   DATA[560,19] := 2.0;
   DATA[560,20] := 148.808;
   DATA[560,21] := 156.0369;
   DATA[560,22] := 1.722487;
   DATA[560,23] := 988.6696;
   DATA[560,24] := 2.0;
   DATA[560,25] := 2.0;
   DATA[560,26] := 7.880544;
   DATA[560,27] := 144.7578;
   DATA[560,28] := 263.4581;
   DATA[560,29] := 12.07383;
   DATA[560,30] := 1.731479;
   DATA[560,31] := 1.287306;
   DATA[560,32] := 0.7353967;
   DATA[560,33] := 0.3080421;
   DATA[560,34] := 2.0;
   DATA[560,35] := 251.2977;
   DATA[560,36] := 1.746067;
   DATA[560,37] := 190.0474;
   DATA[560,38] := 0.000128152;
   DATA[560,39] := 1.0;
   DATA[561,0] := 2.621785;
   DATA[561,1] := 530.344;
   DATA[561,2] := 2.0;
   DATA[561,3] := 2.0;
   DATA[561,4] := 262.1764;
   DATA[561,5] := 8.395475;
   DATA[561,6] := 327.9159;
   DATA[561,7] := 2.4427;
   DATA[561,8] := 2.0;
   DATA[561,9] := 2.0;
   DATA[561,10] := 2.0;
   DATA[561,11] := 19.66835;
   DATA[561,12] := 2.211959;
   DATA[561,13] := 981.4791;
   DATA[561,14] := 1.0;
   DATA[561,15] := 2.0;
   DATA[561,16] := 1.0;
   DATA[561,17] := 1.0;
   DATA[561,18] := 1.0;
   DATA[561,19] := 2.0;
   DATA[561,20] := 148.808;
   DATA[561,21] := 156.0369;
   DATA[561,22] := 1.72159;
   DATA[561,23] := 988.7465;
   DATA[561,24] := 2.0;
   DATA[561,25] := 2.0;
   DATA[561,26] := 7.880544;
   DATA[561,27] := 144.7578;
   DATA[561,28] := 263.4261;
   DATA[561,29] := 12.07383;
   DATA[561,30] := 1.731479;
   DATA[561,31] := 1.274625;
   DATA[561,32] := 0.7353967;
   DATA[561,33] := 0.3087468;
   DATA[561,34] := 2.0;
   DATA[561,35] := 251.2977;
   DATA[561,36] := 1.746067;
   DATA[561,37] := 190.0474;
   DATA[561,38] := 0.000128152;
   DATA[561,39] := 1.0;
   DATA[562,0] := 2.61634;
   DATA[562,1] := 531.9534;
   DATA[562,2] := 2.0;
   DATA[562,3] := 2.0;
   DATA[562,4] := 262.1764;
   DATA[562,5] := 8.395475;
   DATA[562,6] := 327.9159;
   DATA[562,7] := 2.4427;
   DATA[562,8] := 2.0;
   DATA[562,9] := 2.0;
   DATA[562,10] := 2.0;
   DATA[562,11] := 19.66835;
   DATA[562,12] := 2.214906;
   DATA[562,13] := 981.4391;
   DATA[562,14] := 1.0;
   DATA[562,15] := 2.0;
   DATA[562,16] := 1.0;
   DATA[562,17] := 1.0;
   DATA[562,18] := 1.0;
   DATA[562,19] := 2.0;
   DATA[562,20] := 148.808;
   DATA[562,21] := 156.0369;
   DATA[562,22] := 1.718515;
   DATA[562,23] := 989.0925;
   DATA[562,24] := 2.0;
   DATA[562,25] := 2.0;
   DATA[562,26] := 7.880544;
   DATA[562,27] := 144.7578;
   DATA[562,28] := 263.4261;
   DATA[562,29] := 12.07383;
   DATA[562,30] := 1.731479;
   DATA[562,31] := 1.261432;
   DATA[562,32] := 0.7353967;
   DATA[562,33] := 0.3068891;
   DATA[562,34] := 2.0;
   DATA[562,35] := 251.0734;
   DATA[562,36] := 1.746067;
   DATA[562,37] := 189.727;
   DATA[562,38] := 0.000128152;
   DATA[562,39] := 1.0;
   DATA[563,0] := 2.6157;
   DATA[563,1] := 532.5422;
   DATA[563,2] := 2.0;
   DATA[563,3] := 2.0;
   DATA[563,4] := 262.1764;
   DATA[563,5] := 8.395155;
   DATA[563,6] := 327.9159;
   DATA[563,7] := 2.4427;
   DATA[563,8] := 2.0;
   DATA[563,9] := 2.0;
   DATA[563,10] := 2.0;
   DATA[563,11] := 19.66835;
   DATA[563,12] := 2.214906;
   DATA[563,13] := 981.5593;
   DATA[563,14] := 1.0;
   DATA[563,15] := 2.0;
   DATA[563,16] := 1.0;
   DATA[563,17] := 1.0;
   DATA[563,18] := 1.0;
   DATA[563,19] := 2.0;
   DATA[563,20] := 148.808;
   DATA[563,21] := 156.0369;
   DATA[563,22] := 1.718515;
   DATA[563,23] := 988.708;
   DATA[563,24] := 2.0;
   DATA[563,25] := 2.0;
   DATA[563,26] := 7.880544;
   DATA[563,27] := 144.7578;
   DATA[563,28] := 263.4261;
   DATA[563,29] := 12.07383;
   DATA[563,30] := 1.731479;
   DATA[563,31] := 1.25554;
   DATA[563,32] := 0.7353967;
   DATA[563,33] := 0.3066329;
   DATA[563,34] := 2.0;
   DATA[563,35] := 251.0734;
   DATA[563,36] := 1.746067;
   DATA[563,37] := 189.727;
   DATA[563,38] := 0.000128152;
   DATA[563,39] := 1.0;
   DATA[564,0] := 2.593601;
   DATA[564,1] := 532.8954;
   DATA[564,2] := 2.0;
   DATA[564,3] := 2.0;
   DATA[564,4] := 262.1764;
   DATA[564,5] := 8.394835;
   DATA[564,6] := 327.9159;
   DATA[564,7] := 2.444879;
   DATA[564,8] := 2.0;
   DATA[564,9] := 2.0;
   DATA[564,10] := 2.0;
   DATA[564,11] := 19.66835;
   DATA[564,12] := 2.21324;
   DATA[564,13] := 980.8383;
   DATA[564,14] := 1.0;
   DATA[564,15] := 2.0;
   DATA[564,16] := 1.0;
   DATA[564,17] := 1.0;
   DATA[564,18] := 1.0;
   DATA[564,19] := 2.0;
   DATA[564,20] := 148.808;
   DATA[564,21] := 156.0369;
   DATA[564,22] := 1.718515;
   DATA[564,23] := 989.0925;
   DATA[564,24] := 2.0;
   DATA[564,25] := 2.0;
   DATA[564,26] := 7.880544;
   DATA[564,27] := 144.7578;
   DATA[564,28] := 263.4261;
   DATA[564,29] := 12.07383;
   DATA[564,30] := 1.7293;
   DATA[564,31] := 1.254643;
   DATA[564,32] := 0.7353967;
   DATA[564,33] := 0.3065048;
   DATA[564,34] := 2.0;
   DATA[564,35] := 250.9773;
   DATA[564,36] := 1.746067;
   DATA[564,37] := 189.727;
   DATA[564,38] := 0.000128152;
   DATA[564,39] := 1.0;
   DATA[565,0] := 2.572142;
   DATA[565,1] := 532.9739;
   DATA[565,2] := 2.0;
   DATA[565,3] := 2.0;
   DATA[565,4] := 262.1764;
   DATA[565,5] := 8.394835;
   DATA[565,6] := 327.9159;
   DATA[565,7] := 2.444879;
   DATA[565,8] := 2.0;
   DATA[565,9] := 2.0;
   DATA[565,10] := 2.0;
   DATA[565,11] := 19.67796;
   DATA[565,12] := 2.21324;
   DATA[565,13] := 981.1587;
   DATA[565,14] := 1.0;
   DATA[565,15] := 2.0;
   DATA[565,16] := 1.0;
   DATA[565,17] := 1.0;
   DATA[565,18] := 1.0;
   DATA[565,19] := 2.0;
   DATA[565,20] := 148.808;
   DATA[565,21] := 156.0369;
   DATA[565,22] := 1.718515;
   DATA[565,23] := 988.9387;
   DATA[565,24] := 2.0;
   DATA[565,25] := 2.0;
   DATA[565,26] := 7.880544;
   DATA[565,27] := 144.7578;
   DATA[565,28] := 263.4261;
   DATA[565,29] := 12.07383;
   DATA[565,30] := 1.7293;
   DATA[565,31] := 1.268989;
   DATA[565,32] := 0.7353967;
   DATA[565,33] := 0.3065048;
   DATA[565,34] := 2.0;
   DATA[565,35] := 250.9132;
   DATA[565,36] := 1.746067;
   DATA[565,37] := 189.5988;
   DATA[565,38] := 0.000128152;
   DATA[565,39] := 1.0;
   DATA[566,0] := 2.560933;
   DATA[566,1] := 532.8562;
   DATA[566,2] := 2.0;
   DATA[566,3] := 2.0;
   DATA[566,4] := 262.1764;
   DATA[566,5] := 8.394835;
   DATA[566,6] := 327.9159;
   DATA[566,7] := 2.444879;
   DATA[566,8] := 2.0;
   DATA[566,9] := 2.0;
   DATA[566,10] := 2.0;
   DATA[566,11] := 19.67796;
   DATA[566,12] := 2.21324;
   DATA[566,13] := 981.1987;
   DATA[566,14] := 1.0;
   DATA[566,15] := 2.0;
   DATA[566,16] := 1.0;
   DATA[566,17] := 1.0;
   DATA[566,18] := 1.0;
   DATA[566,19] := 2.0;
   DATA[566,20] := 148.808;
   DATA[566,21] := 156.0369;
   DATA[566,22] := 1.717105;
   DATA[566,23] := 988.4773;
   DATA[566,24] := 2.0;
   DATA[566,25] := 2.0;
   DATA[566,26] := 7.880544;
   DATA[566,27] := 144.7578;
   DATA[566,28] := 263.4261;
   DATA[566,29] := 12.07383;
   DATA[566,30] := 1.726096;
   DATA[566,31] := 1.271039;
   DATA[566,32] := 0.736421;
   DATA[566,33] := 0.3065048;
   DATA[566,34] := 2.0;
   DATA[566,35] := 250.5928;
   DATA[566,36] := 1.665972;
   DATA[566,37] := 189.5347;
   DATA[566,38] := 0.000128152;
   DATA[566,39] := 1.0;
   DATA[567,0] := 2.542036;
   DATA[567,1] := 532.7384;
   DATA[567,2] := 2.0;
   DATA[567,3] := 2.0;
   DATA[567,4] := 262.1764;
   DATA[567,5] := 8.394835;
   DATA[567,6] := 327.9159;
   DATA[567,7] := 2.442444;
   DATA[567,8] := 2.0;
   DATA[567,9] := 2.0;
   DATA[567,10] := 2.0;
   DATA[567,11] := 19.67796;
   DATA[567,12] := 2.21324;
   DATA[567,13] := 981.1587;
   DATA[567,14] := 1.0;
   DATA[567,15] := 2.0;
   DATA[567,16] := 1.0;
   DATA[567,17] := 1.0;
   DATA[567,18] := 1.0;
   DATA[567,19] := 2.0;
   DATA[567,20] := 148.808;
   DATA[567,21] := 156.0369;
   DATA[567,22] := 1.716592;
   DATA[567,23] := 989.0541;
   DATA[567,24] := 2.0;
   DATA[567,25] := 2.0;
   DATA[567,26] := 7.880544;
   DATA[567,27] := 144.8859;
   DATA[567,28] := 263.4261;
   DATA[567,29] := 12.07383;
   DATA[567,30] := 1.726096;
   DATA[567,31] := 1.280261;
   DATA[567,32] := 0.7370611;
   DATA[567,33] := 0.3065048;
   DATA[567,34] := 2.0;
   DATA[567,35] := 250.5928;
   DATA[567,36] := 1.665972;
   DATA[567,37] := 189.5027;
   DATA[567,38] := 0.000128152;
   DATA[567,39] := 1.0;
   DATA[568,0] := 2.530506;
   DATA[568,1] := 532.4637;
   DATA[568,2] := 2.0;
   DATA[568,3] := 2.0;
   DATA[568,4] := 262.1764;
   DATA[568,5] := 8.394835;
   DATA[568,6] := 327.9159;
   DATA[568,7] := 2.441162;
   DATA[568,8] := 2.0;
   DATA[568,9] := 2.0;
   DATA[568,10] := 2.0;
   DATA[568,11] := 19.63954;
   DATA[568,12] := 2.211318;
   DATA[568,13] := 980.9985;
   DATA[568,14] := 1.0;
   DATA[568,15] := 2.0;
   DATA[568,16] := 1.0;
   DATA[568,17] := 1.0;
   DATA[568,18] := 1.0;
   DATA[568,19] := 2.0;
   DATA[568,20] := 148.808;
   DATA[568,21] := 156.0369;
   DATA[568,22] := 1.716592;
   DATA[568,23] := 988.708;
   DATA[568,24] := 2.0;
   DATA[568,25] := 2.0;
   DATA[568,26] := 7.880544;
   DATA[568,27] := 144.9116;
   DATA[568,28] := 263.4261;
   DATA[568,29] := 12.07383;
   DATA[568,30] := 1.726096;
   DATA[568,31] := 1.290124;
   DATA[568,32] := 0.7370611;
   DATA[568,33] := 0.3083624;
   DATA[568,34] := 2.0;
   DATA[568,35] := 250.5928;
   DATA[568,36] := 1.665972;
   DATA[568,37] := 189.5027;
   DATA[568,38] := 0.000128152;
   DATA[568,39] := 1.0;
   DATA[569,0] := 2.510649;
   DATA[569,1] := 532.2674;
   DATA[569,2] := 2.0;
   DATA[569,3] := 2.0;
   DATA[569,4] := 262.1764;
   DATA[569,5] := 8.394835;
   DATA[569,6] := 327.9159;
   DATA[569,7] := 2.440521;
   DATA[569,8] := 2.0;
   DATA[569,9] := 2.0;
   DATA[569,10] := 2.0;
   DATA[569,11] := 19.63954;
   DATA[569,12] := 2.210294;
   DATA[569,13] := 980.638;
   DATA[569,14] := 1.0;
   DATA[569,15] := 2.0;
   DATA[569,16] := 1.0;
   DATA[569,17] := 1.0;
   DATA[569,18] := 1.0;
   DATA[569,19] := 2.0;
   DATA[569,20] := 148.808;
   DATA[569,21] := 156.0369;
   DATA[569,22] := 1.717746;
   DATA[569,23] := 988.8618;
   DATA[569,24] := 2.0;
   DATA[569,25] := 2.0;
   DATA[569,26] := 7.880544;
   DATA[569,27] := 144.9116;
   DATA[569,28] := 263.4261;
   DATA[569,29] := 12.07383;
   DATA[569,30] := 1.726096;
   DATA[569,31] := 1.291277;
   DATA[569,32] := 0.7370611;
   DATA[569,33] := 0.3083624;
   DATA[569,34] := 2.0;
   DATA[569,35] := 250.8171;
   DATA[569,36] := 1.665972;
   DATA[569,37] := 189.5027;
   DATA[569,38] := 0.000128152;
   DATA[569,39] := 1.0;
   DATA[570,0] := 2.498799;
   DATA[570,1] := 532.3459;
   DATA[570,2] := 2.0;
   DATA[570,3] := 2.0;
   DATA[570,4] := 262.1764;
   DATA[570,5] := 8.394835;
   DATA[570,6] := 327.9159;
   DATA[570,7] := 2.439881;
   DATA[570,8] := 2.0;
   DATA[570,9] := 2.0;
   DATA[570,10] := 2.0;
   DATA[570,11] := 19.63954;
   DATA[570,12] := 2.210294;
   DATA[570,13] := 980.598;
   DATA[570,14] := 1.0;
   DATA[570,15] := 2.0;
   DATA[570,16] := 1.0;
   DATA[570,17] := 1.0;
   DATA[570,18] := 1.0;
   DATA[570,19] := 2.0;
   DATA[570,20] := 148.808;
   DATA[570,21] := 156.0369;
   DATA[570,22] := 1.717746;
   DATA[570,23] := 988.8618;
   DATA[570,24] := 2.0;
   DATA[570,25] := 2.0;
   DATA[570,26] := 7.880544;
   DATA[570,27] := 144.9116;
   DATA[570,28] := 263.4261;
   DATA[570,29] := 12.07383;
   DATA[570,30] := 1.726096;
   DATA[570,31] := 1.286025;
   DATA[570,32] := 0.7359089;
   DATA[570,33] := 0.3083624;
   DATA[570,34] := 2.0;
   DATA[570,35] := 250.8652;
   DATA[570,36] := 1.665972;
   DATA[570,37] := 189.5027;
   DATA[570,38] := 0.000128152;
   DATA[570,39] := 1.0;
   DATA[571,0] := 2.484066;
   DATA[571,1] := 532.1497;
   DATA[571,2] := 2.0;
   DATA[571,3] := 2.0;
   DATA[571,4] := 262.1764;
   DATA[571,5] := 8.394835;
   DATA[571,6] := 327.9159;
   DATA[571,7] := 2.439881;
   DATA[571,8] := 2.0;
   DATA[571,9] := 2.0;
   DATA[571,10] := 2.0;
   DATA[571,11] := 19.65875;
   DATA[571,12] := 2.214777;
   DATA[571,13] := 980.638;
   DATA[571,14] := 1.0;
   DATA[571,15] := 2.0;
   DATA[571,16] := 1.0;
   DATA[571,17] := 1.0;
   DATA[571,18] := 1.0;
   DATA[571,19] := 2.0;
   DATA[571,20] := 148.808;
   DATA[571,21] := 156.0369;
   DATA[571,22] := 1.717746;
   DATA[571,23] := 989.4386;
   DATA[571,24] := 2.0;
   DATA[571,25] := 2.0;
   DATA[571,26] := 7.880544;
   DATA[571,27] := 144.9116;
   DATA[571,28] := 263.4261;
   DATA[571,29] := 12.07383;
   DATA[571,30] := 1.726096;
   DATA[571,31] := 1.287947;
   DATA[571,32] := 0.7347566;
   DATA[571,33] := 0.3083624;
   DATA[571,34] := 2.0;
   DATA[571,35] := 250.9453;
   DATA[571,36] := 1.665972;
   DATA[571,37] := 189.743;
   DATA[571,38] := 0.000128152;
   DATA[571,39] := 1.0;
   DATA[572,0] := 2.475098;
   DATA[572,1] := 532.0711;
   DATA[572,2] := 2.0;
   DATA[572,3] := 2.0;
   DATA[572,4] := 262.1764;
   DATA[572,5] := 8.394835;
   DATA[572,6] := 327.9159;
   DATA[572,7] := 2.439881;
   DATA[572,8] := 2.0;
   DATA[572,9] := 2.0;
   DATA[572,10] := 2.0;
   DATA[572,11] := 19.65875;
   DATA[572,12] := 2.214777;
   DATA[572,13] := 980.5579;
   DATA[572,14] := 1.0;
   DATA[572,15] := 2.0;
   DATA[572,16] := 1.0;
   DATA[572,17] := 1.0;
   DATA[572,18] := 1.0;
   DATA[572,19] := 2.0;
   DATA[572,20] := 148.808;
   DATA[572,21] := 155.8575;
   DATA[572,22] := 1.717746;
   DATA[572,23] := 989.131;
   DATA[572,24] := 2.0;
   DATA[572,25] := 2.0;
   DATA[572,26] := 7.880544;
   DATA[572,27] := 144.9116;
   DATA[572,28] := 263.4261;
   DATA[572,29] := 12.07383;
   DATA[572,30] := 1.726352;
   DATA[572,31] := 1.272064;
   DATA[572,32] := 0.7347566;
   DATA[572,33] := 0.3083624;
   DATA[572,34] := 2.0;
   DATA[572,35] := 250.9453;
   DATA[572,36] := 1.665972;
   DATA[572,37] := 189.743;
   DATA[572,38] := 0.000128152;
   DATA[572,39] := 1.0;
   DATA[573,0] := 2.462287;
   DATA[573,1] := 531.7964;
   DATA[573,2] := 2.0;
   DATA[573,3] := 2.0;
   DATA[573,4] := 262.1764;
   DATA[573,5] := 8.394835;
   DATA[573,6] := 327.9159;
   DATA[573,7] := 2.439881;
   DATA[573,8] := 2.0;
   DATA[573,9] := 2.0;
   DATA[573,10] := 2.0;
   DATA[573,11] := 19.70037;
   DATA[573,12] := 2.21324;
   DATA[573,13] := 980.7982;
   DATA[573,14] := 1.0;
   DATA[573,15] := 2.0;
   DATA[573,16] := 1.0;
   DATA[573,17] := 1.0;
   DATA[573,18] := 1.0;
   DATA[573,19] := 2.0;
   DATA[573,20] := 148.808;
   DATA[573,21] := 155.8575;
   DATA[573,22] := 1.717746;
   DATA[573,23] := 989.4001;
   DATA[573,24] := 2.0;
   DATA[573,25] := 2.0;
   DATA[573,26] := 7.880544;
   DATA[573,27] := 144.9116;
   DATA[573,28] := 263.4261;
   DATA[573,29] := 12.07383;
   DATA[573,30] := 1.726737;
   DATA[573,31] := 1.280005;
   DATA[573,32] := 0.7347566;
   DATA[573,33] := 0.3083624;
   DATA[573,34] := 2.0;
   DATA[573,35] := 250.9453;
   DATA[573,36] := 1.665972;
   DATA[573,37] := 189.743;
   DATA[573,38] := 0.000128152;
   DATA[573,39] := 1.0;
   DATA[574,0] := 2.449476;
   DATA[574,1] := 531.9141;
   DATA[574,2] := 2.0;
   DATA[574,3] := 2.0;
   DATA[574,4] := 262.1764;
   DATA[574,5] := 8.394835;
   DATA[574,6] := 327.839;
   DATA[574,7] := 2.442188;
   DATA[574,8] := 2.0;
   DATA[574,9] := 2.0;
   DATA[574,10] := 2.0;
   DATA[574,11] := 19.70037;
   DATA[574,12] := 2.212215;
   DATA[574,13] := 980.7982;
   DATA[574,14] := 1.0;
   DATA[574,15] := 2.0;
   DATA[574,16] := 1.0;
   DATA[574,17] := 1.0;
   DATA[574,18] := 1.0;
   DATA[574,19] := 2.0;
   DATA[574,20] := 148.808;
   DATA[574,21] := 155.8575;
   DATA[574,22] := 1.717746;
   DATA[574,23] := 989.3232;
   DATA[574,24] := 2.0;
   DATA[574,25] := 2.0;
   DATA[574,26] := 7.880544;
   DATA[574,27] := 144.9116;
   DATA[574,28] := 263.4261;
   DATA[574,29] := 12.07383;
   DATA[574,30] := 1.726737;
   DATA[574,31] := 1.291405;
   DATA[574,32] := 0.7347566;
   DATA[574,33] := 0.3083624;
   DATA[574,34] := 2.0;
   DATA[574,35] := 250.9453;
   DATA[574,36] := 1.665972;
   DATA[574,37] := 189.743;
   DATA[574,38] := 0.000128152;
   DATA[574,39] := 1.0;
   DATA[575,0] := 2.433142;
   DATA[575,1] := 532.1889;
   DATA[575,2] := 2.0;
   DATA[575,3] := 2.0;
   DATA[575,4] := 262.1764;
   DATA[575,5] := 8.394835;
   DATA[575,6] := 327.839;
   DATA[575,7] := 2.442188;
   DATA[575,8] := 2.0;
   DATA[575,9] := 2.0;
   DATA[575,10] := 2.0;
   DATA[575,11] := 19.73878;
   DATA[575,12] := 2.212215;
   DATA[575,13] := 980.678;
   DATA[575,14] := 1.0;
   DATA[575,15] := 2.0;
   DATA[575,16] := 1.0;
   DATA[575,17] := 1.0;
   DATA[575,18] := 1.0;
   DATA[575,19] := 2.0;
   DATA[575,20] := 148.808;
   DATA[575,21] := 155.678;
   DATA[575,22] := 1.717746;
   DATA[575,23] := 989.4771;
   DATA[575,24] := 2.0;
   DATA[575,25] := 2.0;
   DATA[575,26] := 7.880544;
   DATA[575,27] := 144.9116;
   DATA[575,28] := 263.4261;
   DATA[575,29] := 12.07383;
   DATA[575,30] := 1.728531;
   DATA[575,31] := 1.291405;
   DATA[575,32] := 0.7355248;
   DATA[575,33] := 0.3083624;
   DATA[575,34] := 2.0;
   DATA[575,35] := 250.9773;
   DATA[575,36] := 1.665972;
   DATA[575,37] := 189.743;
   DATA[575,38] := 0.000128152;
   DATA[575,39] := 1.0;
   DATA[576,0] := 2.428979;
   DATA[576,1] := 532.3459;
   DATA[576,2] := 2.0;
   DATA[576,3] := 2.0;
   DATA[576,4] := 262.1764;
   DATA[576,5] := 8.394835;
   DATA[576,6] := 327.839;
   DATA[576,7] := 2.442188;
   DATA[576,8] := 2.0;
   DATA[576,9] := 2.0;
   DATA[576,10] := 2.0;
   DATA[576,11] := 19.74838;
   DATA[576,12] := 2.21055;
   DATA[576,13] := 980.598;
   DATA[576,14] := 1.0;
   DATA[576,15] := 2.0;
   DATA[576,16] := 1.0;
   DATA[576,17] := 1.0;
   DATA[576,18] := 1.0;
   DATA[576,19] := 2.0;
   DATA[576,20] := 148.808;
   DATA[576,21] := 155.678;
   DATA[576,22] := 1.717746;
   DATA[576,23] := 989.5155;
   DATA[576,24] := 2.0;
   DATA[576,25] := 2.0;
   DATA[576,26] := 7.880544;
   DATA[576,27] := 144.9116;
   DATA[576,28] := 263.4261;
   DATA[576,29] := 12.07383;
   DATA[576,30] := 1.728531;
   DATA[576,31] := 1.291405;
   DATA[576,32] := 0.7355248;
   DATA[576,33] := 0.3083624;
   DATA[576,34] := 2.0;
   DATA[576,35] := 250.9933;
   DATA[576,36] := 1.665972;
   DATA[576,37] := 189.743;
   DATA[576,38] := 0.000128152;
   DATA[576,39] := 1.0;
   DATA[577,0] := 2.428979;
   DATA[577,1] := 532.6992;
   DATA[577,2] := 2.0;
   DATA[577,3] := 2.0;
   DATA[577,4] := 262.1764;
   DATA[577,5] := 8.394835;
   DATA[577,6] := 327.839;
   DATA[577,7] := 2.442188;
   DATA[577,8] := 2.0;
   DATA[577,9] := 2.0;
   DATA[577,10] := 2.0;
   DATA[577,11] := 19.74838;
   DATA[577,12] := 2.209525;
   DATA[577,13] := 980.7582;
   DATA[577,14] := 1.0;
   DATA[577,15] := 2.0;
   DATA[577,16] := 1.0;
   DATA[577,17] := 1.0;
   DATA[577,18] := 1.0;
   DATA[577,19] := 2.0;
   DATA[577,20] := 148.808;
   DATA[577,21] := 155.678;
   DATA[577,22] := 1.717746;
   DATA[577,23] := 989.7847;
   DATA[577,24] := 2.0;
   DATA[577,25] := 2.0;
   DATA[577,26] := 7.880544;
   DATA[577,27] := 144.9116;
   DATA[577,28] := 263.3299;
   DATA[577,29] := 12.07383;
   DATA[577,30] := 1.728531;
   DATA[577,31] := 1.280902;
   DATA[577,32] := 0.7355248;
   DATA[577,33] := 0.3083624;
   DATA[577,34] := 2.0;
   DATA[577,35] := 250.9933;
   DATA[577,36] := 1.665972;
   DATA[577,37] := 189.743;
   DATA[577,38] := 0.000128152;
   DATA[577,39] := 1.0;
   DATA[578,0] := 2.458444;
   DATA[578,1] := 532.7384;
   DATA[578,2] := 2.0;
   DATA[578,3] := 2.0;
   DATA[578,4] := 262.1764;
   DATA[578,5] := 8.394835;
   DATA[578,6] := 327.839;
   DATA[578,7] := 2.44411;
   DATA[578,8] := 2.0;
   DATA[578,9] := 2.0;
   DATA[578,10] := 2.0;
   DATA[578,11] := 19.74838;
   DATA[578,12] := 2.207475;
   DATA[578,13] := 980.8383;
   DATA[578,14] := 1.0;
   DATA[578,15] := 2.0;
   DATA[578,16] := 1.0;
   DATA[578,17] := 1.0;
   DATA[578,18] := 1.0;
   DATA[578,19] := 2.0;
   DATA[578,20] := 148.808;
   DATA[578,21] := 155.678;
   DATA[578,22] := 1.717746;
   DATA[578,23] := 989.8616;
   DATA[578,24] := 2.0;
   DATA[578,25] := 2.0;
   DATA[578,26] := 7.880544;
   DATA[578,27] := 144.9116;
   DATA[578,28] := 263.3299;
   DATA[578,29] := 12.07383;
   DATA[578,30] := 1.728531;
   DATA[578,31] := 1.263097;
   DATA[578,32] := 0.7355248;
   DATA[578,33] := 0.3083624;
   DATA[578,34] := 2.0;
   DATA[578,35] := 250.9933;
   DATA[578,36] := 1.665972;
   DATA[578,37] := 189.743;
   DATA[578,38] := 0.000128152;
   DATA[578,39] := 1.0;
   DATA[579,0] := 2.495596;
   DATA[579,1] := 533.3272;
   DATA[579,2] := 2.0;
   DATA[579,3] := 2.0;
   DATA[579,4] := 262.1764;
   DATA[579,5] := 8.394835;
   DATA[579,6] := 327.839;
   DATA[579,7] := 2.442956;
   DATA[579,8] := 2.0;
   DATA[579,9] := 2.0;
   DATA[579,10] := 2.0;
   DATA[579,11] := 19.74838;
   DATA[579,12] := 2.206066;
   DATA[579,13] := 981.0786;
   DATA[579,14] := 1.0;
   DATA[579,15] := 2.0;
   DATA[579,16] := 1.0;
   DATA[579,17] := 1.0;
   DATA[579,18] := 1.0;
   DATA[579,19] := 2.0;
   DATA[579,20] := 148.808;
   DATA[579,21] := 155.678;
   DATA[579,22] := 1.715952;
   DATA[579,23] := 989.7847;
   DATA[579,24] := 2.0;
   DATA[579,25] := 2.0;
   DATA[579,26] := 7.880544;
   DATA[579,27] := 144.9116;
   DATA[579,28] := 263.3299;
   DATA[579,29] := 12.07383;
   DATA[579,30] := 1.728531;
   DATA[579,31] := 1.261816;
   DATA[579,32] := 0.7355248;
   DATA[579,33] := 0.3083624;
   DATA[579,34] := 2.0;
   DATA[579,35] := 250.9933;
   DATA[579,36] := 1.778105;
   DATA[579,37] := 189.743;
   DATA[579,38] := 0.000128152;
   DATA[579,39] := 1.0;
   DATA[580,0] := 2.535311;
   DATA[580,1] := 533.5235;
   DATA[580,2] := 2.0;
   DATA[580,3] := 2.0;
   DATA[580,4] := 262.1764;
   DATA[580,5] := 8.394835;
   DATA[580,6] := 327.9672;
   DATA[580,7] := 2.440906;
   DATA[580,8] := 2.0;
   DATA[580,9] := 2.0;
   DATA[580,10] := 2.0;
   DATA[580,11] := 19.74838;
   DATA[580,12] := 2.208884;
   DATA[580,13] := 981.2388;
   DATA[580,14] := 1.0;
   DATA[580,15] := 2.0;
   DATA[580,16] := 1.0;
   DATA[580,17] := 1.0;
   DATA[580,18] := 1.0;
   DATA[580,19] := 2.0;
   DATA[580,20] := 148.808;
   DATA[580,21] := 155.678;
   DATA[580,22] := 1.715952;
   DATA[580,23] := 990.4384;
   DATA[580,24] := 2.0;
   DATA[580,25] := 2.0;
   DATA[580,26] := 7.880544;
   DATA[580,27] := 145.0397;
   DATA[580,28] := 263.3299;
   DATA[580,29] := 12.07383;
   DATA[580,30] := 1.728531;
   DATA[580,31] := 1.270911;
   DATA[580,32] := 0.7355248;
   DATA[580,33] := 0.3083624;
   DATA[580,34] := 2.0;
   DATA[580,35] := 250.8011;
   DATA[580,36] := 1.778105;
   DATA[580,37] := 189.6789;
   DATA[580,38] := 0.000128152;
   DATA[580,39] := 1.0;
   DATA[581,0] := 2.571182;
   DATA[581,1] := 533.4843;
   DATA[581,2] := 2.0;
   DATA[581,3] := 2.0;
   DATA[581,4] := 262.1764;
   DATA[581,5] := 8.394835;
   DATA[581,6] := 327.9672;
   DATA[581,7] := 2.438984;
   DATA[581,8] := 2.0;
   DATA[581,9] := 2.0;
   DATA[581,10] := 2.0;
   DATA[581,11] := 19.85082;
   DATA[581,12] := 2.208884;
   DATA[581,13] := 981.2789;
   DATA[581,14] := 1.0;
   DATA[581,15] := 2.0;
   DATA[581,16] := 1.0;
   DATA[581,17] := 1.0;
   DATA[581,18] := 1.0;
   DATA[581,19] := 2.0;
   DATA[581,20] := 148.808;
   DATA[581,21] := 155.678;
   DATA[581,22] := 1.713389;
   DATA[581,23] := 990.2461;
   DATA[581,24] := 2.0;
   DATA[581,25] := 2.0;
   DATA[581,26] := 7.880544;
   DATA[581,27] := 145.0397;
   DATA[581,28] := 263.3299;
   DATA[581,29] := 12.07383;
   DATA[581,30] := 1.728531;
   DATA[581,31] := 1.288587;
   DATA[581,32] := 0.7355248;
   DATA[581,33] := 0.3083624;
   DATA[581,34] := 2.0;
   DATA[581,35] := 250.8011;
   DATA[581,36] := 1.778105;
   DATA[581,37] := 189.6148;
   DATA[581,38] := 0.000128152;
   DATA[581,39] := 1.0;
   DATA[582,0] := 2.571182;
   DATA[582,1] := 533.4843;
   DATA[582,2] := 2.0;
   DATA[582,3] := 2.0;
   DATA[582,4] := 262.1764;
   DATA[582,5] := 8.394835;
   DATA[582,6] := 327.9672;
   DATA[582,7] := 2.438984;
   DATA[582,8] := 2.0;
   DATA[582,9] := 2.0;
   DATA[582,10] := 2.0;
   DATA[582,11] := 19.85082;
   DATA[582,12] := 2.208884;
   DATA[582,13] := 981.2789;
   DATA[582,14] := 1.0;
   DATA[582,15] := 2.0;
   DATA[582,16] := 1.0;
   DATA[582,17] := 1.0;
   DATA[582,18] := 1.0;
   DATA[582,19] := 2.0;
   DATA[582,20] := 148.808;
   DATA[582,21] := 155.678;
   DATA[582,22] := 1.713389;
   DATA[582,23] := 990.2461;
   DATA[582,24] := 2.0;
   DATA[582,25] := 2.0;
   DATA[582,26] := 7.880544;
   DATA[582,27] := 145.0397;
   DATA[582,28] := 263.3299;
   DATA[582,29] := 12.07383;
   DATA[582,30] := 1.728531;
   DATA[582,31] := 1.288587;
   DATA[582,32] := 0.7355248;
   DATA[582,33] := 0.3083624;
   DATA[582,34] := 2.0;
   DATA[582,35] := 250.8011;
   DATA[582,36] := 1.778105;
   DATA[582,37] := 189.6148;
   DATA[582,38] := 0.000128152;
   DATA[582,39] := 1.0;
   DATA[583,0] := 2.60417;
   DATA[583,1] := 533.131;
   DATA[583,2] := 2.0;
   DATA[583,3] := 2.0;
   DATA[583,4] := 262.1764;
   DATA[583,5] := 8.394835;
   DATA[583,6] := 327.9672;
   DATA[583,7] := 2.438984;
   DATA[583,8] := 2.0;
   DATA[583,9] := 2.0;
   DATA[583,10] := 2.0;
   DATA[583,11] := 19.85082;
   DATA[583,12] := 2.208884;
   DATA[583,13] := 981.0786;
   DATA[583,14] := 1.0;
   DATA[583,15] := 2.0;
   DATA[583,16] := 1.0;
   DATA[583,17] := 1.0;
   DATA[583,18] := 1.0;
   DATA[583,19] := 2.0;
   DATA[583,20] := 148.808;
   DATA[583,21] := 155.678;
   DATA[583,22] := 1.713261;
   DATA[583,23] := 990.0154;
   DATA[583,24] := 2.0;
   DATA[583,25] := 2.0;
   DATA[583,26] := 7.880544;
   DATA[583,27] := 145.0397;
   DATA[583,28] := 263.3299;
   DATA[583,29] := 12.07383;
   DATA[583,30] := 1.728531;
   DATA[583,31] := 1.300372;
   DATA[583,32] := 0.7355248;
   DATA[583,33] := 0.3083624;
   DATA[583,34] := 2.0;
   DATA[583,35] := 250.8011;
   DATA[583,36] := 1.649953;
   DATA[583,37] := 189.6148;
   DATA[583,38] := 0.000128152;
   DATA[583,39] := 1.0;
   DATA[584,0] := 2.628831;
   DATA[584,1] := 533.3272;
   DATA[584,2] := 2.0;
   DATA[584,3] := 2.0;
   DATA[584,4] := 262.1764;
   DATA[584,5] := 8.394835;
   DATA[584,6] := 327.9672;
   DATA[584,7] := 2.438984;
   DATA[584,8] := 2.0;
   DATA[584,9] := 2.0;
   DATA[584,10] := 2.0;
   DATA[584,11] := 19.85082;
   DATA[584,12] := 2.208884;
   DATA[584,13] := 981.7595;
   DATA[584,14] := 1.0;
   DATA[584,15] := 2.0;
   DATA[584,16] := 1.0;
   DATA[584,17] := 1.0;
   DATA[584,18] := 1.0;
   DATA[584,19] := 2.0;
   DATA[584,20] := 148.808;
   DATA[584,21] := 155.678;
   DATA[584,22] := 1.713261;
   DATA[584,23] := 990.0923;
   DATA[584,24] := 2.0;
   DATA[584,25] := 2.0;
   DATA[584,26] := 7.880544;
   DATA[584,27] := 145.0397;
   DATA[584,28] := 263.3299;
   DATA[584,29] := 12.15073;
   DATA[584,30] := 1.726609;
   DATA[584,31] := 1.30114;
   DATA[584,32] := 0.7355248;
   DATA[584,33] := 0.3083624;
   DATA[584,34] := 2.0;
   DATA[584,35] := 250.8011;
   DATA[584,36] := 1.649953;
   DATA[584,37] := 189.6148;
   DATA[584,38] := 0.000128152;
   DATA[584,39] := 1.0;
   DATA[585,0] := 2.647407;
   DATA[585,1] := 533.445;
   DATA[585,2] := 2.0;
   DATA[585,3] := 2.0;
   DATA[585,4] := 262.1764;
   DATA[585,5] := 8.394835;
   DATA[585,6] := 327.9672;
   DATA[585,7] := 2.440137;
   DATA[585,8] := 2.0;
   DATA[585,9] := 2.0;
   DATA[585,10] := 2.0;
   DATA[585,11] := 19.85082;
   DATA[585,12] := 2.208884;
   DATA[585,13] := 981.8396;
   DATA[585,14] := 1.0;
   DATA[585,15] := 2.0;
   DATA[585,16] := 1.0;
   DATA[585,17] := 1.0;
   DATA[585,18] := 1.0;
   DATA[585,19] := 2.0;
   DATA[585,20] := 148.808;
   DATA[585,21] := 155.678;
   DATA[585,22] := 1.712363;
   DATA[585,23] := 990.0154;
   DATA[585,24] := 2.0;
   DATA[585,25] := 2.0;
   DATA[585,26] := 7.880544;
   DATA[585,27] := 145.0397;
   DATA[585,28] := 263.3299;
   DATA[585,29] := 12.15073;
   DATA[585,30] := 1.724814;
   DATA[585,31] := 1.30114;
   DATA[585,32] := 0.7355248;
   DATA[585,33] := 0.3083624;
   DATA[585,34] := 2.0;
   DATA[585,35] := 250.6729;
   DATA[585,36] := 1.649953;
   DATA[585,37] := 189.5187;
   DATA[585,38] := 0.000128152;
   DATA[585,39] := 1.0;
   DATA[586,0] := 2.64997;
   DATA[586,1] := 533.1702;
   DATA[586,2] := 2.0;
   DATA[586,3] := 2.0;
   DATA[586,4] := 262.1764;
   DATA[586,5] := 8.394835;
   DATA[586,6] := 327.9672;
   DATA[586,7] := 2.440521;
   DATA[586,8] := 2.0;
   DATA[586,9] := 2.0;
   DATA[586,10] := 2.0;
   DATA[586,11] := 19.85082;
   DATA[586,12] := 2.208884;
   DATA[586,13] := 982.2802;
   DATA[586,14] := 1.0;
   DATA[586,15] := 2.0;
   DATA[586,16] := 1.0;
   DATA[586,17] := 1.0;
   DATA[586,18] := 1.0;
   DATA[586,19] := 2.0;
   DATA[586,20] := 148.808;
   DATA[586,21] := 155.678;
   DATA[586,22] := 1.712363;
   DATA[586,23] := 990.0154;
   DATA[586,24] := 2.0;
   DATA[586,25] := 2.0;
   DATA[586,26] := 7.880544;
   DATA[586,27] := 145.0397;
   DATA[586,28] := 263.3299;
   DATA[586,29] := 12.15073;
   DATA[586,30] := 1.724814;
   DATA[586,31] := 1.285513;
   DATA[586,32] := 0.7355248;
   DATA[586,33] := 0.3083624;
   DATA[586,34] := 2.0;
   DATA[586,35] := 250.5127;
   DATA[586,36] := 1.649953;
   DATA[586,37] := 189.3745;
   DATA[586,38] := 0.000128152;
   DATA[586,39] := 1.0;
   DATA[587,0] := 2.632034;
   DATA[587,1] := 533.1702;
   DATA[587,2] := 2.0;
   DATA[587,3] := 2.0;
   DATA[587,4] := 262.1764;
   DATA[587,5] := 8.394835;
   DATA[587,6] := 327.9672;
   DATA[587,7] := 2.440521;
   DATA[587,8] := 2.0;
   DATA[587,9] := 2.0;
   DATA[587,10] := 2.0;
   DATA[587,11] := 19.8028;
   DATA[587,12] := 2.208884;
   DATA[587,13] := 982.7609;
   DATA[587,14] := 1.0;
   DATA[587,15] := 2.0;
   DATA[587,16] := 1.0;
   DATA[587,17] := 1.0;
   DATA[587,18] := 1.0;
   DATA[587,19] := 2.0;
   DATA[587,20] := 148.808;
   DATA[587,21] := 155.7037;
   DATA[587,22] := 1.712363;
   DATA[587,23] := 990.1692;
   DATA[587,24] := 2.0;
   DATA[587,25] := 2.0;
   DATA[587,26] := 7.880544;
   DATA[587,27] := 145.0397;
   DATA[587,28] := 263.3299;
   DATA[587,29] := 12.15073;
   DATA[587,30] := 1.724814;
   DATA[587,31] := 1.282823;
   DATA[587,32] := 0.7355248;
   DATA[587,33] := 0.3083624;
   DATA[587,34] := 2.0;
   DATA[587,35] := 250.5127;
   DATA[587,36] := 1.649953;
   DATA[587,37] := 189.3745;
   DATA[587,38] := 0.000128152;
   DATA[587,39] := 1.0;
   DATA[588,0] := 2.621145;
   DATA[588,1] := 533.3665;
   DATA[588,2] := 2.0;
   DATA[588,3] := 2.0;
   DATA[588,4] := 262.1764;
   DATA[588,5] := 8.394835;
   DATA[588,6] := 327.9672;
   DATA[588,7] := 2.440521;
   DATA[588,8] := 2.0;
   DATA[588,9] := 2.0;
   DATA[588,10] := 2.0;
   DATA[588,11] := 19.8028;
   DATA[588,12] := 2.208884;
   DATA[588,13] := 983.1614;
   DATA[588,14] := 1.0;
   DATA[588,15] := 2.0;
   DATA[588,16] := 1.0;
   DATA[588,17] := 1.0;
   DATA[588,18] := 1.0;
   DATA[588,19] := 2.0;
   DATA[588,20] := 148.808;
   DATA[588,21] := 155.7293;
   DATA[588,22] := 1.714542;
   DATA[588,23] := 990.3615;
   DATA[588,24] := 2.0;
   DATA[588,25] := 2.0;
   DATA[588,26] := 7.880544;
   DATA[588,27] := 145.0397;
   DATA[588,28] := 263.3299;
   DATA[588,29] := 12.15073;
   DATA[588,30] := 1.724814;
   DATA[588,31] := 1.287691;
   DATA[588,32] := 0.7355248;
   DATA[588,33] := 0.3083624;
   DATA[588,34] := 2.0;
   DATA[588,35] := 250.5127;
   DATA[588,36] := 1.649953;
   DATA[588,37] := 189.3745;
   DATA[588,38] := 0.000128152;
   DATA[588,39] := 1.0;
   DATA[589,0] := 2.613138;
   DATA[589,1] := 533.0917;
   DATA[589,2] := 2.0;
   DATA[589,3] := 2.0;
   DATA[589,4] := 262.1764;
   DATA[589,5] := 8.394835;
   DATA[589,6] := 327.9672;
   DATA[589,7] := 2.440521;
   DATA[589,8] := 2.0;
   DATA[589,9] := 2.0;
   DATA[589,10] := 2.0;
   DATA[589,11] := 19.84442;
   DATA[589,12] := 2.208884;
   DATA[589,13] := 983.4818;
   DATA[589,14] := 1.0;
   DATA[589,15] := 2.0;
   DATA[589,16] := 1.0;
   DATA[589,17] := 1.0;
   DATA[589,18] := 1.0;
   DATA[589,19] := 2.0;
   DATA[589,20] := 148.808;
   DATA[589,21] := 155.7293;
   DATA[589,22] := 1.714542;
   DATA[589,23] := 990.4768;
   DATA[589,24] := 2.0;
   DATA[589,25] := 2.0;
   DATA[589,26] := 7.880544;
   DATA[589,27] := 145.0397;
   DATA[589,28] := 263.3299;
   DATA[589,29] := 12.15073;
   DATA[589,30] := 1.724814;
   DATA[589,31] := 1.282951;
   DATA[589,32] := 0.7355248;
   DATA[589,33] := 0.3083624;
   DATA[589,34] := 2.0;
   DATA[589,35] := 250.5127;
   DATA[589,36] := 1.649953;
   DATA[589,37] := 189.3745;
   DATA[589,38] := 0.000128152;
   DATA[589,39] := 1.0;
   DATA[590,0] := 2.605131;
   DATA[590,1] := 533.0524;
   DATA[590,2] := 2.0;
   DATA[590,3] := 2.0;
   DATA[590,4] := 262.1764;
   DATA[590,5] := 8.394835;
   DATA[590,6] := 327.9672;
   DATA[590,7] := 2.441162;
   DATA[590,8] := 2.0;
   DATA[590,9] := 2.0;
   DATA[590,10] := 2.0;
   DATA[590,11] := 19.84442;
   DATA[590,12] := 2.208884;
   DATA[590,13] := 983.8423;
   DATA[590,14] := 1.0;
   DATA[590,15] := 2.0;
   DATA[590,16] := 1.0;
   DATA[590,17] := 1.0;
   DATA[590,18] := 1.0;
   DATA[590,19] := 2.0;
   DATA[590,20] := 148.808;
   DATA[590,21] := 155.7293;
   DATA[590,22] := 1.714542;
   DATA[590,23] := 990.2845;
   DATA[590,24] := 2.0;
   DATA[590,25] := 2.0;
   DATA[590,26] := 7.880544;
   DATA[590,27] := 145.0397;
   DATA[590,28] := 263.3299;
   DATA[590,29] := 12.15073;
   DATA[590,30] := 1.724814;
   DATA[590,31] := 1.27296;
   DATA[590,32] := 0.7355248;
   DATA[590,33] := 0.3083624;
   DATA[590,34] := 2.0;
   DATA[590,35] := 250.5127;
   DATA[590,36] := 1.649953;
   DATA[590,37] := 189.3745;
   DATA[590,38] := 0.000128152;
   DATA[590,39] := 1.0;
   DATA[591,0] := 2.588156;
   DATA[591,1] := 532.8954;
   DATA[591,2] := 2.0;
   DATA[591,3] := 2.0;
   DATA[591,4] := 262.1764;
   DATA[591,5] := 8.394835;
   DATA[591,6] := 327.6596;
   DATA[591,7] := 2.441162;
   DATA[591,8] := 2.0;
   DATA[591,9] := 2.0;
   DATA[591,10] := 2.0;
   DATA[591,11] := 19.77399;
   DATA[591,12] := 2.208884;
   DATA[591,13] := 984.4031;
   DATA[591,14] := 1.0;
   DATA[591,15] := 2.0;
   DATA[591,16] := 1.0;
   DATA[591,17] := 1.0;
   DATA[591,18] := 1.0;
   DATA[591,19] := 2.0;
   DATA[591,20] := 148.808;
   DATA[591,21] := 155.7293;
   DATA[591,22] := 1.714542;
   DATA[591,23] := 990.5537;
   DATA[591,24] := 2.0;
   DATA[591,25] := 2.0;
   DATA[591,26] := 7.880544;
   DATA[591,27] := 145.0397;
   DATA[591,28] := 263.3299;
   DATA[591,29] := 12.15073;
   DATA[591,30] := 1.724045;
   DATA[591,31] := 1.271423;
   DATA[591,32] := 0.7355248;
   DATA[591,33] := 0.3083624;
   DATA[591,34] := 2.0;
   DATA[591,35] := 250.5127;
   DATA[591,36] := 1.649953;
   DATA[591,37] := 189.3745;
   DATA[591,38] := 0.000128152;
   DATA[591,39] := 1.0;
   DATA[592,0] := 2.56958;
   DATA[592,1] := 532.6599;
   DATA[592,2] := 2.0;
   DATA[592,3] := 2.0;
   DATA[592,4] := 262.1764;
   DATA[592,5] := 8.394835;
   DATA[592,6] := 327.6596;
   DATA[592,7] := 2.441162;
   DATA[592,8] := 2.0;
   DATA[592,9] := 2.0;
   DATA[592,10] := 2.0;
   DATA[592,11] := 19.72598;
   DATA[592,12] := 2.208884;
   DATA[592,13] := 985.0038;
   DATA[592,14] := 1.0;
   DATA[592,15] := 2.0;
   DATA[592,16] := 1.0;
   DATA[592,17] := 1.0;
   DATA[592,18] := 1.0;
   DATA[592,19] := 2.0;
   DATA[592,20] := 148.808;
   DATA[592,21] := 155.7293;
   DATA[592,22] := 1.715439;
   DATA[592,23] := 990.3999;
   DATA[592,24] := 2.0;
   DATA[592,25] := 2.0;
   DATA[592,26] := 7.880544;
   DATA[592,27] := 145.0397;
   DATA[592,28] := 263.3299;
   DATA[592,29] := 12.15073;
   DATA[592,30] := 1.724045;
   DATA[592,31] := 1.273345;
   DATA[592,32] := 0.7355248;
   DATA[592,33] := 0.3083624;
   DATA[592,34] := 2.0;
   DATA[592,35] := 250.5127;
   DATA[592,36] := 1.649953;
   DATA[592,37] := 189.3745;
   DATA[592,38] := 0.000128152;
   DATA[592,39] := 1.0;
   DATA[593,0] := 2.556129;
   DATA[593,1] := 532.3851;
   DATA[593,2] := 2.0;
   DATA[593,3] := 2.0;
   DATA[593,4] := 262.1764;
   DATA[593,5] := 8.396116;
   DATA[593,6] := 327.6596;
   DATA[593,7] := 2.439753;
   DATA[593,8] := 2.0;
   DATA[593,9] := 2.0;
   DATA[593,10] := 2.0;
   DATA[593,11] := 19.72598;
   DATA[593,12] := 2.208884;
   DATA[593,13] := 985.1641;
   DATA[593,14] := 1.0;
   DATA[593,15] := 2.0;
   DATA[593,16] := 1.0;
   DATA[593,17] := 1.0;
   DATA[593,18] := 1.0;
   DATA[593,19] := 2.0;
   DATA[593,20] := 148.808;
   DATA[593,21] := 155.7293;
   DATA[593,22] := 1.715439;
   DATA[593,23] := 990.746;
   DATA[593,24] := 2.0;
   DATA[593,25] := 2.0;
   DATA[593,26] := 7.880544;
   DATA[593,27] := 145.0397;
   DATA[593,28] := 263.1377;
   DATA[593,29] := 12.15073;
   DATA[593,30] := 1.724045;
   DATA[593,31] := 1.277699;
   DATA[593,32] := 0.7355248;
   DATA[593,33] := 0.3083624;
   DATA[593,34] := 2.0;
   DATA[593,35] := 250.5127;
   DATA[593,36] := 1.649953;
   DATA[593,37] := 189.3745;
   DATA[593,38] := 0.000128152;
   DATA[593,39] := 1.0;
   DATA[594,0] := 2.542677;
   DATA[594,1] := 532.1104;
   DATA[594,2] := 2.0;
   DATA[594,3] := 2.0;
   DATA[594,4] := 262.1764;
   DATA[594,5] := 8.396116;
   DATA[594,6] := 327.6596;
   DATA[594,7] := 2.439753;
   DATA[594,8] := 2.0;
   DATA[594,9] := 2.0;
   DATA[594,10] := 2.0;
   DATA[594,11] := 19.66195;
   DATA[594,12] := 2.208884;
   DATA[594,13] := 985.6848;
   DATA[594,14] := 1.0;
   DATA[594,15] := 2.0;
   DATA[594,16] := 1.0;
   DATA[594,17] := 1.0;
   DATA[594,18] := 1.0;
   DATA[594,19] := 2.0;
   DATA[594,20] := 148.808;
   DATA[594,21] := 155.7293;
   DATA[594,22] := 1.717105;
   DATA[594,23] := 990.4384;
   DATA[594,24] := 2.0;
   DATA[594,25] := 2.0;
   DATA[594,26] := 7.880544;
   DATA[594,27] := 145.0397;
   DATA[594,28] := 263.1377;
   DATA[594,29] := 12.15073;
   DATA[594,30] := 1.726352;
   DATA[594,31] := 1.272576;
   DATA[594,32] := 0.7355248;
   DATA[594,33] := 0.3083624;
   DATA[594,34] := 2.0;
   DATA[594,35] := 250.5928;
   DATA[594,36] := 1.649953;
   DATA[594,37] := 189.3745;
   DATA[594,38] := 0.000128152;
   DATA[594,39] := 1.0;
   DATA[595,0] := 2.521218;
   DATA[595,1] := 532.1104;
   DATA[595,2] := 2.0;
   DATA[595,3] := 2.0;
   DATA[595,4] := 262.1764;
   DATA[595,5] := 8.396116;
   DATA[595,6] := 327.8647;
   DATA[595,7] := 2.439753;
   DATA[595,8] := 2.0;
   DATA[595,9] := 2.0;
   DATA[595,10] := 2.0;
   DATA[595,11] := 19.65555;
   DATA[595,12] := 2.209013;
   DATA[595,13] := 986.2055;
   DATA[595,14] := 1.0;
   DATA[595,15] := 2.0;
   DATA[595,16] := 1.0;
   DATA[595,17] := 1.0;
   DATA[595,18] := 1.0;
   DATA[595,19] := 2.0;
   DATA[595,20] := 148.808;
   DATA[595,21] := 155.7293;
   DATA[595,22] := 1.717361;
   DATA[595,23] := 990.4384;
   DATA[595,24] := 2.0;
   DATA[595,25] := 2.0;
   DATA[595,26] := 7.880544;
   DATA[595,27] := 145.0397;
   DATA[595,28] := 263.1377;
   DATA[595,29] := 12.15073;
   DATA[595,30] := 1.726993;
   DATA[595,31] := 1.25823;
   DATA[595,32] := 0.7355248;
   DATA[595,33] := 0.3083624;
   DATA[595,34] := 2.0;
   DATA[595,35] := 250.753;
   DATA[595,36] := 1.649953;
   DATA[595,37] := 189.3745;
   DATA[595,38] := 0.000128152;
   DATA[595,39] := 1.0;
   DATA[596,0] := 2.508728;
   DATA[596,1] := 531.6001;
   DATA[596,2] := 2.0;
   DATA[596,3] := 2.0;
   DATA[596,4] := 262.1764;
   DATA[596,5] := 8.396116;
   DATA[596,6] := 327.8647;
   DATA[596,7] := 2.442188;
   DATA[596,8] := 2.0;
   DATA[596,9] := 2.0;
   DATA[596,10] := 2.0;
   DATA[596,11] := 19.65555;
   DATA[596,12] := 2.209909;
   DATA[596,13] := 986.1654;
   DATA[596,14] := 1.0;
   DATA[596,15] := 2.0;
   DATA[596,16] := 1.0;
   DATA[596,17] := 1.0;
   DATA[596,18] := 1.0;
   DATA[596,19] := 2.0;
   DATA[596,20] := 148.808;
   DATA[596,21] := 155.7293;
   DATA[596,22] := 1.717361;
   DATA[596,23] := 990.6306;
   DATA[596,24] := 2.0;
   DATA[596,25] := 2.0;
   DATA[596,26] := 7.880544;
   DATA[596,27] := 145.0397;
   DATA[596,28] := 263.1377;
   DATA[596,29] := 12.15073;
   DATA[596,30] := 1.726993;
   DATA[596,31] := 1.254515;
   DATA[596,32] := 0.7355248;
   DATA[596,33] := 0.3083624;
   DATA[596,34] := 2.0;
   DATA[596,35] := 250.753;
   DATA[596,36] := 1.649953;
   DATA[596,37] := 189.4066;
   DATA[596,38] := 0.000128152;
   DATA[596,39] := 1.0;
   DATA[597,0] := 2.48823;
   DATA[597,1] := 531.9534;
   DATA[597,2] := 2.0;
   DATA[597,3] := 2.0;
   DATA[597,4] := 262.1764;
   DATA[597,5] := 8.396116;
   DATA[597,6] := 327.8647;
   DATA[597,7] := 2.442188;
   DATA[597,8] := 2.0;
   DATA[597,9] := 2.0;
   DATA[597,10] := 2.0;
   DATA[597,11] := 19.65555;
   DATA[597,12] := 2.212343;
   DATA[597,13] := 986.0853;
   DATA[597,14] := 1.0;
   DATA[597,15] := 2.0;
   DATA[597,16] := 1.0;
   DATA[597,17] := 1.0;
   DATA[597,18] := 1.0;
   DATA[597,19] := 2.0;
   DATA[597,20] := 148.808;
   DATA[597,21] := 155.7293;
   DATA[597,22] := 1.717361;
   DATA[597,23] := 990.5922;
   DATA[597,24] := 2.0;
   DATA[597,25] := 2.0;
   DATA[597,26] := 7.880544;
   DATA[597,27] := 145.0397;
   DATA[597,28] := 263.1377;
   DATA[597,29] := 12.15073;
   DATA[597,30] := 1.726993;
   DATA[597,31] := 1.258102;
   DATA[597,32] := 0.7355248;
   DATA[597,33] := 0.3083624;
   DATA[597,34] := 2.0;
   DATA[597,35] := 250.8171;
   DATA[597,36] := 1.649953;
   DATA[597,37] := 189.6629;
   DATA[597,38] := 0.000128152;
   DATA[597,39] := 1.0;
   DATA[598,0] := 2.47702;
   DATA[598,1] := 532.3066;
   DATA[598,2] := 2.0;
   DATA[598,3] := 2.0;
   DATA[598,4] := 262.1764;
   DATA[598,5] := 8.396116;
   DATA[598,6] := 327.8647;
   DATA[598,7] := 2.440137;
   DATA[598,8] := 2.0;
   DATA[598,9] := 2.0;
   DATA[598,10] := 2.0;
   DATA[598,11] := 19.70677;
   DATA[598,12] := 2.212343;
   DATA[598,13] := 986.0052;
   DATA[598,14] := 1.0;
   DATA[598,15] := 2.0;
   DATA[598,16] := 1.0;
   DATA[598,17] := 1.0;
   DATA[598,18] := 1.0;
   DATA[598,19] := 2.0;
   DATA[598,20] := 148.808;
   DATA[598,21] := 155.7806;
   DATA[598,22] := 1.718387;
   DATA[598,23] := 990.8229;
   DATA[598,24] := 2.0;
   DATA[598,25] := 2.0;
   DATA[598,26] := 7.880544;
   DATA[598,27] := 145.0397;
   DATA[598,28] := 263.1377;
   DATA[598,29] := 12.15073;
   DATA[598,30] := 1.726993;
   DATA[598,31] := 1.278468;
   DATA[598,32] := 0.7355248;
   DATA[598,33] := 0.3083624;
   DATA[598,34] := 2.0;
   DATA[598,35] := 250.8972;
   DATA[598,36] := 1.649953;
   DATA[598,37] := 189.6789;
   DATA[598,38] := 0.000128152;
   DATA[598,39] := 1.0;
   DATA[599,0] := 2.460045;
   DATA[599,1] := 533.1702;
   DATA[599,2] := 2.0;
   DATA[599,3] := 2.0;
   DATA[599,4] := 262.1764;
   DATA[599,5] := 8.396116;
   DATA[599,6] := 327.8647;
   DATA[599,7] := 2.439625;
   DATA[599,8] := 2.0;
   DATA[599,9] := 2.0;
   DATA[599,10] := 2.0;
   DATA[599,11] := 19.71637;
   DATA[599,12] := 2.212343;
   DATA[599,13] := 986.3657;
   DATA[599,14] := 1.0;
   DATA[599,15] := 2.0;
   DATA[599,16] := 1.0;
   DATA[599,17] := 1.0;
   DATA[599,18] := 1.0;
   DATA[599,19] := 2.0;
   DATA[599,20] := 148.808;
   DATA[599,21] := 155.7806;
   DATA[599,22] := 1.719156;
   DATA[599,23] := 990.9382;
   DATA[599,24] := 2.0;
   DATA[599,25] := 2.0;
   DATA[599,26] := 7.880544;
   DATA[599,27] := 145.0397;
   DATA[599,28] := 263.1377;
   DATA[599,29] := 12.15073;
   DATA[599,30] := 1.728019;
   DATA[599,31] := 1.297682;
   DATA[599,32] := 0.7355248;
   DATA[599,33] := 0.3083624;
   DATA[599,34] := 2.0;
   DATA[599,35] := 250.8972;
   DATA[599,36] := 1.649953;
   DATA[599,37] := 189.6789;
   DATA[599,38] := 0.000128152;
   DATA[599,39] := 1.0;
   DATA[600,0] := 2.446594;
   DATA[600,1] := 533.759;
   DATA[600,2] := 2.0;
   DATA[600,3] := 2.0;
   DATA[600,4] := 262.1764;
   DATA[600,5] := 8.396116;
   DATA[600,6] := 327.8647;
   DATA[600,7] := 2.439625;
   DATA[600,8] := 2.0;
   DATA[600,9] := 2.0;
   DATA[600,10] := 2.0;
   DATA[600,11] := 19.67155;
   DATA[600,12] := 2.212343;
   DATA[600,13] := 986.6461;
   DATA[600,14] := 1.0;
   DATA[600,15] := 2.0;
   DATA[600,16] := 1.0;
   DATA[600,17] := 1.0;
   DATA[600,18] := 1.0;
   DATA[600,19] := 2.0;
   DATA[600,20] := 148.808;
   DATA[600,21] := 155.7806;
   DATA[600,22] := 1.720565;
   DATA[600,23] := 990.9382;
   DATA[600,24] := 2.0;
   DATA[600,25] := 2.0;
   DATA[600,26] := 7.880544;
   DATA[600,27] := 145.0397;
   DATA[600,28] := 263.1377;
   DATA[600,29] := 12.15073;
   DATA[600,30] := 1.728659;
   DATA[600,31] := 1.297169;
   DATA[600,32] := 0.7355248;
   DATA[600,33] := 0.3075937;
   DATA[600,34] := 2.0;
   DATA[600,35] := 250.8972;
   DATA[600,36] := 1.649953;
   DATA[600,37] := 189.6789;
   DATA[600,38] := 0.000128152;
   DATA[600,39] := 1.0;
   DATA[601,0] := 2.433783;
   DATA[601,1] := 534.3085;
   DATA[601,2] := 2.0;
   DATA[601,3] := 2.0;
   DATA[601,4] := 262.1764;
   DATA[601,5] := 8.396116;
   DATA[601,6] := 327.8647;
   DATA[601,7] := 2.439625;
   DATA[601,8] := 2.0;
   DATA[601,9] := 2.0;
   DATA[601,10] := 2.0;
   DATA[601,11] := 19.67155;
   DATA[601,12] := 2.212343;
   DATA[601,13] := 987.0065;
   DATA[601,14] := 1.0;
   DATA[601,15] := 2.0;
   DATA[601,16] := 1.0;
   DATA[601,17] := 1.0;
   DATA[601,18] := 1.0;
   DATA[601,19] := 2.0;
   DATA[601,20] := 148.808;
   DATA[601,21] := 155.7806;
   DATA[601,22] := 1.720565;
   DATA[601,23] := 990.7844;
   DATA[601,24] := 2.0;
   DATA[601,25] := 2.0;
   DATA[601,26] := 7.880544;
   DATA[601,27] := 145.0397;
   DATA[601,28] := 263.1377;
   DATA[601,29] := 12.15073;
   DATA[601,30] := 1.728659;
   DATA[601,31] := 1.282823;
   DATA[601,32] := 0.7355248;
   DATA[601,33] := 0.3070813;
   DATA[601,34] := 2.0;
   DATA[601,35] := 250.8972;
   DATA[601,36] := 1.649953;
   DATA[601,37] := 189.6789;
   DATA[601,38] := 0.000128152;
   DATA[601,39] := 1.0;
   DATA[602,0] := 2.426737;
   DATA[602,1] := 534.5441;
   DATA[602,2] := 2.0;
   DATA[602,3] := 2.0;
   DATA[602,4] := 262.1764;
   DATA[602,5] := 8.396116;
   DATA[602,6] := 327.8647;
   DATA[602,7] := 2.439625;
   DATA[602,8] := 2.0;
   DATA[602,9] := 2.0;
   DATA[602,10] := 2.0;
   DATA[602,11] := 19.69396;
   DATA[602,12] := 2.212343;
   DATA[602,13] := 986.9665;
   DATA[602,14] := 1.0;
   DATA[602,15] := 2.0;
   DATA[602,16] := 1.0;
   DATA[602,17] := 1.0;
   DATA[602,18] := 1.0;
   DATA[602,19] := 2.0;
   DATA[602,20] := 148.808;
   DATA[602,21] := 155.7806;
   DATA[602,22] := 1.719156;
   DATA[602,23] := 991.0151;
   DATA[602,24] := 2.0;
   DATA[602,25] := 2.0;
   DATA[602,26] := 7.880544;
   DATA[602,27] := 145.0397;
   DATA[602,28] := 263.1377;
   DATA[602,29] := 12.15073;
   DATA[602,30] := 1.728659;
   DATA[602,31] := 1.281542;
   DATA[602,32] := 0.7355248;
   DATA[602,33] := 0.3063127;
   DATA[602,34] := 2.0;
   DATA[602,35] := 251.0254;
   DATA[602,36] := 1.649953;
   DATA[602,37] := 189.6949;
   DATA[602,38] := 0.000128152;
   DATA[602,39] := 1.0;
   DATA[603,0] := 2.426737;
   DATA[603,1] := 534.7403;
   DATA[603,2] := 2.0;
   DATA[603,3] := 2.0;
   DATA[603,4] := 262.1764;
   DATA[603,5] := 8.396116;
   DATA[603,6] := 327.8647;
   DATA[603,7] := 2.439625;
   DATA[603,8] := 2.0;
   DATA[603,9] := 2.0;
   DATA[603,10] := 2.0;
   DATA[603,11] := 19.69396;
   DATA[603,12] := 2.212343;
   DATA[603,13] := 986.6461;
   DATA[603,14] := 1.0;
   DATA[603,15] := 2.0;
   DATA[603,16] := 1.0;
   DATA[603,17] := 1.0;
   DATA[603,18] := 1.0;
   DATA[603,19] := 2.0;
   DATA[603,20] := 148.808;
   DATA[603,21] := 155.7806;
   DATA[603,22] := 1.716849;
   DATA[603,23] := 990.9382;
   DATA[603,24] := 2.0;
   DATA[603,25] := 2.0;
   DATA[603,26] := 7.880544;
   DATA[603,27] := 145.0397;
   DATA[603,28] := 263.1377;
   DATA[603,29] := 12.15073;
   DATA[603,30] := 1.728659;
   DATA[603,31] := 1.27296;
   DATA[603,32] := 0.7355248;
   DATA[603,33] := 0.3063127;
   DATA[603,34] := 2.0;
   DATA[603,35] := 251.0254;
   DATA[603,36] := 1.649953;
   DATA[603,37] := 189.759;
   DATA[603,38] := 0.000128152;
   DATA[603,39] := 1.0;
   DATA[604,0] := 2.452679;
   DATA[604,1] := 534.8973;
   DATA[604,2] := 2.0;
   DATA[604,3] := 2.0;
   DATA[604,4] := 262.1764;
   DATA[604,5] := 8.396116;
   DATA[604,6] := 327.8647;
   DATA[604,7] := 2.440137;
   DATA[604,8] := 2.0;
   DATA[604,9] := 2.0;
   DATA[604,10] := 2.0;
   DATA[604,11] := 19.69396;
   DATA[604,12] := 2.212343;
   DATA[604,13] := 986.6862;
   DATA[604,14] := 1.0;
   DATA[604,15] := 2.0;
   DATA[604,16] := 1.0;
   DATA[604,17] := 1.0;
   DATA[604,18] := 1.0;
   DATA[604,19] := 2.0;
   DATA[604,20] := 148.808;
   DATA[604,21] := 155.7806;
   DATA[604,22] := 1.716849;
   DATA[604,23] := 991.1689;
   DATA[604,24] := 2.0;
   DATA[604,25] := 2.0;
   DATA[604,26] := 7.880544;
   DATA[604,27] := 145.0397;
   DATA[604,28] := 263.1377;
   DATA[604,29] := 12.15073;
   DATA[604,30] := 1.728659;
   DATA[604,31] := 1.277443;
   DATA[604,32] := 0.7355248;
   DATA[604,33] := 0.3063127;
   DATA[604,34] := 2.0;
   DATA[604,35] := 251.0254;
   DATA[604,36] := 1.649953;
   DATA[604,37] := 189.759;
   DATA[604,38] := 0.000128152;
   DATA[604,39] := 1.0;
   DATA[605,0] := 2.503603;
   DATA[605,1] := 534.9366;
   DATA[605,2] := 2.0;
   DATA[605,3] := 2.0;
   DATA[605,4] := 262.1764;
   DATA[605,5] := 8.396116;
   DATA[605,6] := 327.8647;
   DATA[605,7] := 2.440137;
   DATA[605,8] := 2.0;
   DATA[605,9] := 2.0;
   DATA[605,10] := 2.0;
   DATA[605,11] := 19.69396;
   DATA[605,12] := 2.211575;
   DATA[605,13] := 986.7662;
   DATA[605,14] := 1.0;
   DATA[605,15] := 2.0;
   DATA[605,16] := 1.0;
   DATA[605,17] := 1.0;
   DATA[605,18] := 1.0;
   DATA[605,19] := 2.0;
   DATA[605,20] := 148.808;
   DATA[605,21] := 155.7806;
   DATA[605,22] := 1.716849;
   DATA[605,23] := 991.1305;
   DATA[605,24] := 2.0;
   DATA[605,25] := 2.0;
   DATA[605,26] := 7.880544;
   DATA[605,27] := 145.1679;
   DATA[605,28] := 263.1377;
   DATA[605,29] := 12.15073;
   DATA[605,30] := 1.728659;
   DATA[605,31] := 1.291918;
   DATA[605,32] := 0.7355248;
   DATA[605,33] := 0.3063127;
   DATA[605,34] := 2.0;
   DATA[605,35] := 251.0254;
   DATA[605,36] := 1.649953;
   DATA[605,37] := 189.759;
   DATA[605,38] := 0.000128152;
   DATA[605,39] := 1.0;
   DATA[606,0] := 2.543638;
   DATA[606,1] := 534.8581;
   DATA[606,2] := 2.0;
   DATA[606,3] := 2.0;
   DATA[606,4] := 262.1764;
   DATA[606,5] := 8.396116;
   DATA[606,6] := 327.8647;
   DATA[606,7] := 2.441675;
   DATA[606,8] := 2.0;
   DATA[606,9] := 2.0;
   DATA[606,10] := 2.0;
   DATA[606,11] := 19.74198;
   DATA[606,12] := 2.209653;
   DATA[606,13] := 986.9665;
   DATA[606,14] := 1.0;
   DATA[606,15] := 2.0;
   DATA[606,16] := 1.0;
   DATA[606,17] := 1.0;
   DATA[606,18] := 1.0;
   DATA[606,19] := 2.0;
   DATA[606,20] := 148.808;
   DATA[606,21] := 155.7806;
   DATA[606,22] := 1.71813;
   DATA[606,23] := 990.9382;
   DATA[606,24] := 2.0;
   DATA[606,25] := 2.0;
   DATA[606,26] := 7.880544;
   DATA[606,27] := 145.1679;
   DATA[606,28] := 263.1377;
   DATA[606,29] := 12.15073;
   DATA[606,30] := 1.726096;
   DATA[606,31] := 1.286282;
   DATA[606,32] := 0.7355248;
   DATA[606,33] := 0.3063127;
   DATA[606,34] := 2.0;
   DATA[606,35] := 251.0254;
   DATA[606,36] := 1.649953;
   DATA[606,37] := 189.759;
   DATA[606,38] := 0.000128152;
   DATA[606,39] := 1.0;
   DATA[607,0] := 2.579509;
   DATA[607,1] := 534.8973;
   DATA[607,2] := 2.0;
   DATA[607,3] := 2.0;
   DATA[607,4] := 262.1764;
   DATA[607,5] := 8.395475;
   DATA[607,6] := 327.8647;
   DATA[607,7] := 2.441803;
   DATA[607,8] := 2.0;
   DATA[607,9] := 2.0;
   DATA[607,10] := 2.0;
   DATA[607,11] := 19.74198;
   DATA[607,12] := 2.209653;
   DATA[607,13] := 986.566;
   DATA[607,14] := 1.0;
   DATA[607,15] := 2.0;
   DATA[607,16] := 1.0;
   DATA[607,17] := 1.0;
   DATA[607,18] := 1.0;
   DATA[607,19] := 2.0;
   DATA[607,20] := 148.808;
   DATA[607,21] := 155.7806;
   DATA[607,22] := 1.719156;
   DATA[607,23] := 991.2074;
   DATA[607,24] := 2.0;
   DATA[607,25] := 2.0;
   DATA[607,26] := 7.880544;
   DATA[607,27] := 145.1679;
   DATA[607,28] := 263.1377;
   DATA[607,29] := 12.15073;
   DATA[607,30] := 1.724173;
   DATA[607,31] := 1.287306;
   DATA[607,32] := 0.7355248;
   DATA[607,33] := 0.3063127;
   DATA[607,34] := 2.0;
   DATA[607,35] := 250.8331;
   DATA[607,36] := 1.649953;
   DATA[607,37] := 189.5988;
   DATA[607,38] := 0.000128152;
   DATA[607,39] := 1.0;
   DATA[608,0] := 2.620504;
   DATA[608,1] := 535.0936;
   DATA[608,2] := 2.0;
   DATA[608,3] := 2.0;
   DATA[608,4] := 262.1764;
   DATA[608,5] := 8.395475;
   DATA[608,6] := 327.8647;
   DATA[608,7] := 2.443341;
   DATA[608,8] := 2.0;
   DATA[608,9] := 2.0;
   DATA[608,10] := 2.0;
   DATA[608,11] := 19.69396;
   DATA[608,12] := 2.209653;
   DATA[608,13] := 986.4458;
   DATA[608,14] := 1.0;
   DATA[608,15] := 2.0;
   DATA[608,16] := 1.0;
   DATA[608,17] := 1.0;
   DATA[608,18] := 1.0;
   DATA[608,19] := 2.0;
   DATA[608,20] := 148.808;
   DATA[608,21] := 155.7806;
   DATA[608,22] := 1.719156;
   DATA[608,23] := 991.5535;
   DATA[608,24] := 2.0;
   DATA[608,25] := 2.0;
   DATA[608,26] := 7.880544;
   DATA[608,27] := 145.1679;
   DATA[608,28] := 263.4261;
   DATA[608,29] := 12.03538;
   DATA[608,30] := 1.724173;
   DATA[608,31] := 1.287691;
   DATA[608,32] := 0.7355248;
   DATA[608,33] := 0.306761;
   DATA[608,34] := 2.0;
   DATA[608,35] := 250.8331;
   DATA[608,36] := 1.649953;
   DATA[608,37] := 189.5988;
   DATA[608,38] := 0.000128152;
   DATA[608,39] := 1.0;
   DATA[609,0] := 2.649009;
   DATA[609,1] := 535.0936;
   DATA[609,2] := 2.0;
   DATA[609,3] := 2.0;
   DATA[609,4] := 262.1764;
   DATA[609,5] := 8.395475;
   DATA[609,6] := 327.8647;
   DATA[609,7] := 2.443597;
   DATA[609,8] := 2.0;
   DATA[609,9] := 2.0;
   DATA[609,10] := 2.0;
   DATA[609,11] := 19.69076;
   DATA[609,12] := 2.209653;
   DATA[609,13] := 986.4458;
   DATA[609,14] := 1.0;
   DATA[609,15] := 2.0;
   DATA[609,16] := 1.0;
   DATA[609,17] := 1.0;
   DATA[609,18] := 1.0;
   DATA[609,19] := 2.0;
   DATA[609,20] := 148.808;
   DATA[609,21] := 155.7806;
   DATA[609,22] := 1.719156;
   DATA[609,23] := 991.7073;
   DATA[609,24] := 2.0;
   DATA[609,25] := 2.0;
   DATA[609,26] := 7.880544;
   DATA[609,27] := 145.1679;
   DATA[609,28] := 263.4261;
   DATA[609,29] := 12.03538;
   DATA[609,30] := 1.725583;
   DATA[609,31] := 1.281158;
   DATA[609,32] := 0.7355248;
   DATA[609,33] := 0.306761;
   DATA[609,34] := 2.0;
   DATA[609,35] := 250.8331;
   DATA[609,36] := 1.649953;
   DATA[609,37] := 189.5988;
   DATA[609,38] := 0.000128152;
   DATA[609,39] := 1.0;
   DATA[610,0] := 2.668225;
   DATA[610,1] := 535.2899;
   DATA[610,2] := 2.0;
   DATA[610,3] := 2.0;
   DATA[610,4] := 262.1764;
   DATA[610,5] := 8.395475;
   DATA[610,6] := 327.8647;
   DATA[610,7] := 2.443597;
   DATA[610,8] := 2.0;
   DATA[610,9] := 2.0;
   DATA[610,10] := 2.0;
   DATA[610,11] := 19.69076;
   DATA[610,12] := 2.209653;
   DATA[610,13] := 986.1654;
   DATA[610,14] := 1.0;
   DATA[610,15] := 2.0;
   DATA[610,16] := 1.0;
   DATA[610,17] := 1.0;
   DATA[610,18] := 1.0;
   DATA[610,19] := 2.0;
   DATA[610,20] := 148.808;
   DATA[610,21] := 155.7806;
   DATA[610,22] := 1.717746;
   DATA[610,23] := 991.9764;
   DATA[610,24] := 2.0;
   DATA[610,25] := 2.0;
   DATA[610,26] := 7.880544;
   DATA[610,27] := 145.1679;
   DATA[610,28] := 263.4261;
   DATA[610,29] := 12.03538;
   DATA[610,30] := 1.725968;
   DATA[610,31] := 1.281158;
   DATA[610,32] := 0.7355248;
   DATA[610,33] := 0.306761;
   DATA[610,34] := 2.0;
   DATA[610,35] := 250.8331;
   DATA[610,36] := 1.649953;
   DATA[610,37] := 189.5988;
   DATA[610,38] := 0.000128152;
   DATA[610,39] := 1.0;
   DATA[611,0] := 2.668225;
   DATA[611,1] := 535.3291;
   DATA[611,2] := 2.0;
   DATA[611,3] := 2.0;
   DATA[611,4] := 262.1764;
   DATA[611,5] := 8.395475;
   DATA[611,6] := 327.8647;
   DATA[611,7] := 2.443597;
   DATA[611,8] := 2.0;
   DATA[611,9] := 2.0;
   DATA[611,10] := 2.0;
   DATA[611,11] := 19.72277;
   DATA[611,12] := 2.209653;
   DATA[611,13] := 986.2055;
   DATA[611,14] := 1.0;
   DATA[611,15] := 2.0;
   DATA[611,16] := 1.0;
   DATA[611,17] := 1.0;
   DATA[611,18] := 1.0;
   DATA[611,19] := 2.0;
   DATA[611,20] := 148.808;
   DATA[611,21] := 155.7806;
   DATA[611,22] := 1.716849;
   DATA[611,23] := 992.3994;
   DATA[611,24] := 2.0;
   DATA[611,25] := 2.0;
   DATA[611,26] := 7.880544;
   DATA[611,27] := 145.1679;
   DATA[611,28] := 263.3299;
   DATA[611,29] := 12.03538;
   DATA[611,30] := 1.726609;
   DATA[611,31] := 1.287947;
   DATA[611,32] := 0.7355248;
   DATA[611,33] := 0.306761;
   DATA[611,34] := 2.0;
   DATA[611,35] := 250.8331;
   DATA[611,36] := 1.649953;
   DATA[611,37] := 189.5988;
   DATA[611,38] := 0.000128152;
   DATA[611,39] := 1.0;
   DATA[612,0] := 2.644525;
   DATA[612,1] := 535.3291;
   DATA[612,2] := 2.0;
   DATA[612,3] := 2.0;
   DATA[612,4] := 262.1764;
   DATA[612,5] := 8.393232;
   DATA[612,6] := 327.8647;
   DATA[612,7] := 2.443597;
   DATA[612,8] := 2.0;
   DATA[612,9] := 2.0;
   DATA[612,10] := 2.0;
   DATA[612,11] := 19.72277;
   DATA[612,12] := 2.21119;
   DATA[612,13] := 986.2055;
   DATA[612,14] := 1.0;
   DATA[612,15] := 2.0;
   DATA[612,16] := 1.0;
   DATA[612,17] := 1.0;
   DATA[612,18] := 1.0;
   DATA[612,19] := 2.0;
   DATA[612,20] := 148.808;
   DATA[612,21] := 155.7806;
   DATA[612,22] := 1.716849;
   DATA[612,23] := 992.5916;
   DATA[612,24] := 2.0;
   DATA[612,25] := 2.0;
   DATA[612,26] := 7.880544;
   DATA[612,27] := 145.1679;
   DATA[612,28] := 263.3299;
   DATA[612,29] := 12.03538;
   DATA[612,30] := 1.727506;
   DATA[612,31] := 1.308441;
   DATA[612,32] := 0.7355248;
   DATA[612,33] := 0.306761;
   DATA[612,34] := 2.0;
   DATA[612,35] := 250.9933;
   DATA[612,36] := 1.649953;
   DATA[612,37] := 189.8231;
   DATA[612,38] := 0.000128152;
   DATA[612,39] := 1.0;
   DATA[613,0] := 2.624347;
   DATA[613,1] := 535.2899;
   DATA[613,2] := 2.0;
   DATA[613,3] := 2.0;
   DATA[613,4] := 262.1764;
   DATA[613,5] := 8.393232;
   DATA[613,6] := 327.8647;
   DATA[613,7] := 2.443725;
   DATA[613,8] := 2.0;
   DATA[613,9] := 2.0;
   DATA[613,10] := 2.0;
   DATA[613,11] := 19.72277;
   DATA[613,12] := 2.21119;
   DATA[613,13] := 985.8851;
   DATA[613,14] := 1.0;
   DATA[613,15] := 2.0;
   DATA[613,16] := 1.0;
   DATA[613,17] := 1.0;
   DATA[613,18] := 1.0;
   DATA[613,19] := 2.0;
   DATA[613,20] := 148.808;
   DATA[613,21] := 155.7806;
   DATA[613,22] := 1.716849;
   DATA[613,23] := 992.5147;
   DATA[613,24] := 2.0;
   DATA[613,25] := 2.0;
   DATA[613,26] := 7.880544;
   DATA[613,27] := 145.1679;
   DATA[613,28] := 263.1697;
   DATA[613,29] := 12.03538;
   DATA[613,30] := 1.727506;
   DATA[613,31] := 1.312412;
   DATA[613,32] := 0.7355248;
   DATA[613,33] := 0.306761;
   DATA[613,34] := 2.0;
   DATA[613,35] := 250.9933;
   DATA[613,36] := 1.649953;
   DATA[613,37] := 189.9353;
   DATA[613,38] := 0.000128152;
   DATA[613,39] := 1.0;
   DATA[614,0] := 2.620824;
   DATA[614,1] := 535.2506;
   DATA[614,2] := 2.0;
   DATA[614,3] := 2.0;
   DATA[614,4] := 262.1764;
   DATA[614,5] := 8.393232;
   DATA[614,6] := 327.8647;
   DATA[614,7] := 2.443725;
   DATA[614,8] := 2.0;
   DATA[614,9] := 2.0;
   DATA[614,10] := 2.0;
   DATA[614,11] := 19.72277;
   DATA[614,12] := 2.21119;
   DATA[614,13] := 985.845;
   DATA[614,14] := 1.0;
   DATA[614,15] := 2.0;
   DATA[614,16] := 1.0;
   DATA[614,17] := 1.0;
   DATA[614,18] := 1.0;
   DATA[614,19] := 2.0;
   DATA[614,20] := 148.808;
   DATA[614,21] := 155.7806;
   DATA[614,22] := 1.716849;
   DATA[614,23] := 992.2841;
   DATA[614,24] := 2.0;
   DATA[614,25] := 2.0;
   DATA[614,26] := 7.880544;
   DATA[614,27] := 145.1679;
   DATA[614,28] := 263.1697;
   DATA[614,29] := 12.03538;
   DATA[614,30] := 1.729813;
   DATA[614,31] := 1.330601;
   DATA[614,32] := 0.7355248;
   DATA[614,33] := 0.306761;
   DATA[614,34] := 2.0;
   DATA[614,35] := 251.0734;
   DATA[614,36] := 1.649953;
   DATA[614,37] := 189.9353;
   DATA[614,38] := 0.000128152;
   DATA[614,39] := 1.0;
   DATA[615,0] := 2.617622;
   DATA[615,1] := 535.4469;
   DATA[615,2] := 2.0;
   DATA[615,3] := 2.0;
   DATA[615,4] := 262.1764;
   DATA[615,5] := 8.394514;
   DATA[615,6] := 327.8647;
   DATA[615,7] := 2.443725;
   DATA[615,8] := 2.0;
   DATA[615,9] := 2.0;
   DATA[615,10] := 2.0;
   DATA[615,11] := 19.72277;
   DATA[615,12] := 2.21119;
   DATA[615,13] := 986.2455;
   DATA[615,14] := 1.0;
   DATA[615,15] := 2.0;
   DATA[615,16] := 1.0;
   DATA[615,17] := 1.0;
   DATA[615,18] := 1.0;
   DATA[615,19] := 2.0;
   DATA[615,20] := 148.808;
   DATA[615,21] := 155.7806;
   DATA[615,22] := 1.716849;
   DATA[615,23] := 992.2841;
   DATA[615,24] := 2.0;
   DATA[615,25] := 2.0;
   DATA[615,26] := 7.880544;
   DATA[615,27] := 145.1679;
   DATA[615,28] := 263.1377;
   DATA[615,29] := 12.03538;
   DATA[615,30] := 1.729813;
   DATA[615,31] := 1.326502;
   DATA[615,32] := 0.7355248;
   DATA[615,33] := 0.306761;
   DATA[615,34] := 2.0;
   DATA[615,35] := 251.2817;
   DATA[615,36] := 1.649953;
   DATA[615,37] := 189.9353;
   DATA[615,38] := 0.000128152;
   DATA[615,39] := 1.0;
   DATA[616,0] := 2.596163;
   DATA[616,1] := 535.4861;
   DATA[616,2] := 2.0;
   DATA[616,3] := 2.0;
   DATA[616,4] := 262.1764;
   DATA[616,5] := 8.394514;
   DATA[616,6] := 327.8647;
   DATA[616,7] := 2.44206;
   DATA[616,8] := 2.0;
   DATA[616,9] := 2.0;
   DATA[616,10] := 2.0;
   DATA[616,11] := 19.72277;
   DATA[616,12] := 2.21119;
   DATA[616,13] := 986.0453;
   DATA[616,14] := 1.0;
   DATA[616,15] := 2.0;
   DATA[616,16] := 1.0;
   DATA[616,17] := 1.0;
   DATA[616,18] := 1.0;
   DATA[616,19] := 2.0;
   DATA[616,20] := 148.808;
   DATA[616,21] := 155.7806;
   DATA[616,22] := 1.717489;
   DATA[616,23] := 992.1687;
   DATA[616,24] := 2.0;
   DATA[616,25] := 2.0;
   DATA[616,26] := 7.880544;
   DATA[616,27] := 145.1679;
   DATA[616,28] := 263.1377;
   DATA[616,29] := 12.03538;
   DATA[616,30] := 1.729813;
   DATA[616,31] := 1.312668;
   DATA[616,32] := 0.7355248;
   DATA[616,33] := 0.306761;
   DATA[616,34] := 2.0;
   DATA[616,35] := 251.2817;
   DATA[616,36] := 1.730048;
   DATA[616,37] := 189.9353;
   DATA[616,38] := 0.000128152;
   DATA[616,39] := 1.0;
   DATA[617,0] := 2.585594;
   DATA[617,1] := 535.3291;
   DATA[617,2] := 2.0;
   DATA[617,3] := 2.0;
   DATA[617,4] := 262.1764;
   DATA[617,5] := 8.394514;
   DATA[617,6] := 327.8647;
   DATA[617,7] := 2.439496;
   DATA[617,8] := 2.0;
   DATA[617,9] := 2.0;
   DATA[617,10] := 2.0;
   DATA[617,11] := 19.66195;
   DATA[617,12] := 2.21119;
   DATA[617,13] := 986.0052;
   DATA[617,14] := 1.0;
   DATA[617,15] := 2.0;
   DATA[617,16] := 1.0;
   DATA[617,17] := 1.0;
   DATA[617,18] := 1.0;
   DATA[617,19] := 2.0;
   DATA[617,20] := 148.808;
   DATA[617,21] := 155.7806;
   DATA[617,22] := 1.717489;
   DATA[617,23] := 992.3994;
   DATA[617,24] := 2.0;
   DATA[617,25] := 2.0;
   DATA[617,26] := 7.880544;
   DATA[617,27] := 145.1679;
   DATA[617,28] := 263.1377;
   DATA[617,29] := 12.03538;
   DATA[617,30] := 1.729813;
   DATA[617,31] := 1.302037;
   DATA[617,32] := 0.7355248;
   DATA[617,33] := 0.306761;
   DATA[617,34] := 2.0;
   DATA[617,35] := 251.2817;
   DATA[617,36] := 1.730048;
   DATA[617,37] := 189.9353;
   DATA[617,38] := 0.000128152;
   DATA[617,39] := 1.0;
   DATA[618,0] := 2.563174;
   DATA[618,1] := 535.6431;
   DATA[618,2] := 2.0;
   DATA[618,3] := 2.0;
   DATA[618,4] := 262.1764;
   DATA[618,5] := 8.394514;
   DATA[618,6] := 327.8647;
   DATA[618,7] := 2.439496;
   DATA[618,8] := 2.0;
   DATA[618,9] := 2.0;
   DATA[618,10] := 2.0;
   DATA[618,11] := 19.66195;
   DATA[618,12] := 2.21119;
   DATA[618,13] := 985.7649;
   DATA[618,14] := 1.0;
   DATA[618,15] := 2.0;
   DATA[618,16] := 1.0;
   DATA[618,17] := 1.0;
   DATA[618,18] := 1.0;
   DATA[618,19] := 2.0;
   DATA[618,20] := 148.808;
   DATA[618,21] := 155.7806;
   DATA[618,22] := 1.719924;
   DATA[618,23] := 992.361;
   DATA[618,24] := 2.0;
   DATA[618,25] := 2.0;
   DATA[618,26] := 7.880544;
   DATA[618,27] := 145.1679;
   DATA[618,28] := 263.1377;
   DATA[618,29] := 12.03538;
   DATA[618,30] := 1.729813;
   DATA[618,31] := 1.291405;
   DATA[618,32] := 0.7355248;
   DATA[618,33] := 0.306761;
   DATA[618,34] := 2.0;
   DATA[618,35] := 251.2817;
   DATA[618,36] := 1.730048;
   DATA[618,37] := 189.9353;
   DATA[618,38] := 0.000128152;
   DATA[618,39] := 1.0;
   DATA[619,0] := 2.547481;
   DATA[619,1] := 535.9179;
   DATA[619,2] := 2.0;
   DATA[619,3] := 2.0;
   DATA[619,4] := 262.1764;
   DATA[619,5] := 8.394514;
   DATA[619,6] := 327.8647;
   DATA[619,7] := 2.439496;
   DATA[619,8] := 2.0;
   DATA[619,9] := 2.0;
   DATA[619,10] := 2.0;
   DATA[619,11] := 19.66195;
   DATA[619,12] := 2.21119;
   DATA[619,13] := 985.6848;
   DATA[619,14] := 1.0;
   DATA[619,15] := 2.0;
   DATA[619,16] := 1.0;
   DATA[619,17] := 1.0;
   DATA[619,18] := 1.0;
   DATA[619,19] := 2.0;
   DATA[619,20] := 148.808;
   DATA[619,21] := 155.7806;
   DATA[619,22] := 1.719924;
   DATA[619,23] := 992.6685;
   DATA[619,24] := 2.0;
   DATA[619,25] := 2.0;
   DATA[619,26] := 7.880544;
   DATA[619,27] := 145.1166;
   DATA[619,28] := 263.1377;
   DATA[619,29] := 12.03538;
   DATA[619,30] := 1.729813;
   DATA[619,31] := 1.280261;
   DATA[619,32] := 0.7355248;
   DATA[619,33] := 0.306761;
   DATA[619,34] := 2.0;
   DATA[619,35] := 251.1215;
   DATA[619,36] := 1.730048;
   DATA[619,37] := 189.9353;
   DATA[619,38] := 0.000128152;
   DATA[619,39] := 1.0;
   DATA[620,0] := 2.525702;
   DATA[620,1] := 536.2712;
   DATA[620,2] := 2.0;
   DATA[620,3] := 2.0;
   DATA[620,4] := 262.1764;
   DATA[620,5] := 8.394514;
   DATA[620,6] := 327.8647;
   DATA[620,7] := 2.439496;
   DATA[620,8] := 2.0;
   DATA[620,9] := 2.0;
   DATA[620,10] := 2.0;
   DATA[620,11] := 19.66195;
   DATA[620,12] := 2.21119;
   DATA[620,13] := 985.4044;
   DATA[620,14] := 1.0;
   DATA[620,15] := 2.0;
   DATA[620,16] := 1.0;
   DATA[620,17] := 1.0;
   DATA[620,18] := 1.0;
   DATA[620,19] := 2.0;
   DATA[620,20] := 148.808;
   DATA[620,21] := 155.7806;
   DATA[620,22] := 1.719924;
   DATA[620,23] := 992.8992;
   DATA[620,24] := 2.0;
   DATA[620,25] := 2.0;
   DATA[620,26] := 7.880544;
   DATA[620,27] := 145.1166;
   DATA[620,28] := 263.1377;
   DATA[620,29] := 12.03538;
   DATA[620,30] := 1.729813;
   DATA[620,31] := 1.271679;
   DATA[620,32] := 0.7355248;
   DATA[620,33] := 0.306761;
   DATA[620,34] := 2.0;
   DATA[620,35] := 251.1215;
   DATA[620,36] := 1.730048;
   DATA[620,37] := 189.8552;
   DATA[620,38] := 0.000128152;
   DATA[620,39] := 1.0;
   DATA[621,0] := 2.510649;
   DATA[621,1] := 536.4675;
   DATA[621,2] := 2.0;
   DATA[621,3] := 2.0;
   DATA[621,4] := 262.1764;
   DATA[621,5] := 8.394514;
   DATA[621,6] := 327.8647;
   DATA[621,7] := 2.441419;
   DATA[621,8] := 2.0;
   DATA[621,9] := 2.0;
   DATA[621,10] := 2.0;
   DATA[621,11] := 19.71637;
   DATA[621,12] := 2.210166;
   DATA[621,13] := 985.8049;
   DATA[621,14] := 1.0;
   DATA[621,15] := 2.0;
   DATA[621,16] := 1.0;
   DATA[621,17] := 1.0;
   DATA[621,18] := 1.0;
   DATA[621,19] := 2.0;
   DATA[621,20] := 148.808;
   DATA[621,21] := 155.7806;
   DATA[621,22] := 1.719924;
   DATA[621,23] := 992.8992;
   DATA[621,24] := 2.0;
   DATA[621,25] := 2.0;
   DATA[621,26] := 7.880544;
   DATA[621,27] := 145.1166;
   DATA[621,28] := 263.1377;
   DATA[621,29] := 12.03538;
   DATA[621,30] := 1.729813;
   DATA[621,31] := 1.271679;
   DATA[621,32] := 0.7355248;
   DATA[621,33] := 0.306761;
   DATA[621,34] := 2.0;
   DATA[621,35] := 251.1215;
   DATA[621,36] := 1.601897;
   DATA[621,37] := 189.8552;
   DATA[621,38] := 0.000128152;
   DATA[621,39] := 1.0;
   DATA[622,0] := 2.491112;
   DATA[622,1] := 536.6637;
   DATA[622,2] := 2.0;
   DATA[622,3] := 2.0;
   DATA[622,4] := 262.1764;
   DATA[622,5] := 8.394514;
   DATA[622,6] := 327.8647;
   DATA[622,7] := 2.441803;
   DATA[622,8] := 2.0;
   DATA[622,9] := 2.0;
   DATA[622,10] := 2.0;
   DATA[622,11] := 19.71637;
   DATA[622,12] := 2.209397;
   DATA[622,13] := 985.7649;
   DATA[622,14] := 1.0;
   DATA[622,15] := 2.0;
   DATA[622,16] := 1.0;
   DATA[622,17] := 1.0;
   DATA[622,18] := 1.0;
   DATA[622,19] := 2.0;
   DATA[622,20] := 148.808;
   DATA[622,21] := 155.7806;
   DATA[622,22] := 1.718771;
   DATA[622,23] := 992.7454;
   DATA[622,24] := 2.0;
   DATA[622,25] := 2.0;
   DATA[622,26] := 7.880544;
   DATA[622,27] := 145.1166;
   DATA[622,28] := 263.1377;
   DATA[622,29] := 12.03538;
   DATA[622,30] := 1.729813;
   DATA[622,31] := 1.261816;
   DATA[622,32] := 0.7355248;
   DATA[622,33] := 0.3075937;
   DATA[622,34] := 2.0;
   DATA[622,35] := 251.1215;
   DATA[622,36] := 1.601897;
   DATA[622,37] := 189.8552;
   DATA[622,38] := 0.000128152;
   DATA[622,39] := 1.0;
   DATA[623,0] := 2.491112;
   DATA[623,1] := 536.6637;
   DATA[623,2] := 2.0;
   DATA[623,3] := 2.0;
   DATA[623,4] := 262.1764;
   DATA[623,5] := 8.394514;
   DATA[623,6] := 327.8647;
   DATA[623,7] := 2.441803;
   DATA[623,8] := 2.0;
   DATA[623,9] := 2.0;
   DATA[623,10] := 2.0;
   DATA[623,11] := 19.71637;
   DATA[623,12] := 2.209397;
   DATA[623,13] := 985.7649;
   DATA[623,14] := 1.0;
   DATA[623,15] := 2.0;
   DATA[623,16] := 1.0;
   DATA[623,17] := 1.0;
   DATA[623,18] := 1.0;
   DATA[623,19] := 2.0;
   DATA[623,20] := 148.808;
   DATA[623,21] := 155.7806;
   DATA[623,22] := 1.718771;
   DATA[623,23] := 992.7454;
   DATA[623,24] := 2.0;
   DATA[623,25] := 2.0;
   DATA[623,26] := 7.880544;
   DATA[623,27] := 145.1166;
   DATA[623,28] := 263.1377;
   DATA[623,29] := 12.03538;
   DATA[623,30] := 1.729813;
   DATA[623,31] := 1.261816;
   DATA[623,32] := 0.7355248;
   DATA[623,33] := 0.3075937;
   DATA[623,34] := 2.0;
   DATA[623,35] := 251.1215;
   DATA[623,36] := 1.601897;
   DATA[623,37] := 189.8552;
   DATA[623,38] := 0.000128152;
   DATA[623,39] := 1.0;
   DATA[624,0] := 2.477661;
   DATA[624,1] := 536.6245;
   DATA[624,2] := 2.0;
   DATA[624,3] := 2.0;
   DATA[624,4] := 262.1764;
   DATA[624,5] := 8.394514;
   DATA[624,6] := 327.8647;
   DATA[624,7] := 2.441803;
   DATA[624,8] := 2.0;
   DATA[624,9] := 2.0;
   DATA[624,10] := 2.0;
   DATA[624,11] := 19.71637;
   DATA[624,12] := 2.209397;
   DATA[624,13] := 985.4845;
   DATA[624,14] := 1.0;
   DATA[624,15] := 2.0;
   DATA[624,16] := 1.0;
   DATA[624,17] := 1.0;
   DATA[624,18] := 1.0;
   DATA[624,19] := 2.0;
   DATA[624,20] := 148.808;
   DATA[624,21] := 155.7806;
   DATA[624,22] := 1.717105;
   DATA[624,23] := 992.7454;
   DATA[624,24] := 2.0;
   DATA[624,25] := 2.0;
   DATA[624,26] := 7.880544;
   DATA[624,27] := 145.1166;
   DATA[624,28] := 263.1377;
   DATA[624,29] := 12.03538;
   DATA[624,30] := 1.729813;
   DATA[624,31] := 1.261048;
   DATA[624,32] := 0.7355248;
   DATA[624,33] := 0.3084265;
   DATA[624,34] := 2.0;
   DATA[624,35] := 251.1215;
   DATA[624,36] := 1.601897;
   DATA[624,37] := 189.8552;
   DATA[624,38] := 0.000128152;
   DATA[624,39] := 1.0;
   DATA[625,0] := 2.460045;
   DATA[625,1] := 536.8207;
   DATA[625,2] := 2.0;
   DATA[625,3] := 2.0;
   DATA[625,4] := 262.1764;
   DATA[625,5] := 8.394514;
   DATA[625,6] := 327.8647;
   DATA[625,7] := 2.440393;
   DATA[625,8] := 2.0;
   DATA[625,9] := 2.0;
   DATA[625,10] := 2.0;
   DATA[625,11] := 19.70357;
   DATA[625,12] := 2.209397;
   DATA[625,13] := 985.6848;
   DATA[625,14] := 1.0;
   DATA[625,15] := 2.0;
   DATA[625,16] := 1.0;
   DATA[625,17] := 1.0;
   DATA[625,18] := 1.0;
   DATA[625,19] := 2.0;
   DATA[625,20] := 148.808;
   DATA[625,21] := 155.7806;
   DATA[625,22] := 1.717105;
   DATA[625,23] := 992.7454;
   DATA[625,24] := 2.0;
   DATA[625,25] := 2.0;
   DATA[625,26] := 7.880544;
   DATA[625,27] := 145.1166;
   DATA[625,28] := 263.1377;
   DATA[625,29] := 12.03538;
   DATA[625,30] := 1.728916;
   DATA[625,31] := 1.261048;
   DATA[625,32] := 0.7355248;
   DATA[625,33] := 0.3084265;
   DATA[625,34] := 2.0;
   DATA[625,35] := 250.8972;
   DATA[625,36] := 1.69801;
   DATA[625,37] := 189.6469;
   DATA[625,38] := 0.000128152;
   DATA[625,39] := 1.0;
   DATA[626,0] := 2.447234;
   DATA[626,1] := 536.86;
   DATA[626,2] := 2.0;
   DATA[626,3] := 2.0;
   DATA[626,4] := 262.1764;
   DATA[626,5] := 8.394514;
   DATA[626,6] := 327.8647;
   DATA[626,7] := 2.439625;
   DATA[626,8] := 2.0;
   DATA[626,9] := 2.0;
   DATA[626,10] := 2.0;
   DATA[626,11] := 19.68756;
   DATA[626,12] := 2.209397;
   DATA[626,13] := 985.6848;
   DATA[626,14] := 1.0;
   DATA[626,15] := 2.0;
   DATA[626,16] := 1.0;
   DATA[626,17] := 1.0;
   DATA[626,18] := 1.0;
   DATA[626,19] := 2.0;
   DATA[626,20] := 148.808;
   DATA[626,21] := 155.7806;
   DATA[626,22] := 1.717105;
   DATA[626,23] := 992.2841;
   DATA[626,24] := 2.0;
   DATA[626,25] := 2.0;
   DATA[626,26] := 7.880544;
   DATA[626,27] := 145.1166;
   DATA[626,28] := 263.1377;
   DATA[626,29] := 12.03538;
   DATA[626,30] := 1.726865;
   DATA[626,31] := 1.272064;
   DATA[626,32] := 0.7355248;
   DATA[626,33] := 0.3084265;
   DATA[626,34] := 2.0;
   DATA[626,35] := 250.8972;
   DATA[626,36] := 1.69801;
   DATA[626,37] := 189.5027;
   DATA[626,38] := 0.000128152;
   DATA[626,39] := 1.0;
   DATA[627,0] := 2.431861;
   DATA[627,1] := 536.9777;
   DATA[627,2] := 2.0;
   DATA[627,3] := 2.0;
   DATA[627,4] := 262.1764;
   DATA[627,5] := 8.394514;
   DATA[627,6] := 327.8647;
   DATA[627,7] := 2.439625;
   DATA[627,8] := 2.0;
   DATA[627,9] := 2.0;
   DATA[627,10] := 2.0;
   DATA[627,11] := 19.68756;
   DATA[627,12] := 2.209397;
   DATA[627,13] := 985.5646;
   DATA[627,14] := 1.0;
   DATA[627,15] := 2.0;
   DATA[627,16] := 1.0;
   DATA[627,17] := 1.0;
   DATA[627,18] := 1.0;
   DATA[627,19] := 2.0;
   DATA[627,20] := 148.808;
   DATA[627,21] := 155.7806;
   DATA[627,22] := 1.717105;
   DATA[627,23] := 992.3994;
   DATA[627,24] := 2.0;
   DATA[627,25] := 2.0;
   DATA[627,26] := 7.880544;
   DATA[627,27] := 145.1166;
   DATA[627,28] := 263.1377;
   DATA[627,29] := 12.03538;
   DATA[627,30] := 1.726865;
   DATA[627,31] := 1.287306;
   DATA[627,32] := 0.7355248;
   DATA[627,33] := 0.3084265;
   DATA[627,34] := 2.0;
   DATA[627,35] := 250.8972;
   DATA[627,36] := 1.69801;
   DATA[627,37] := 189.5027;
   DATA[627,38] := 0.000128152;
   DATA[627,39] := 1.0;
   DATA[628,0] := 2.431861;
   DATA[628,1] := 536.6637;
   DATA[628,2] := 2.0;
   DATA[628,3] := 2.0;
   DATA[628,4] := 262.1764;
   DATA[628,5] := 8.394514;
   DATA[628,6] := 327.7621;
   DATA[628,7] := 2.439625;
   DATA[628,8] := 2.0;
   DATA[628,9] := 2.0;
   DATA[628,10] := 2.0;
   DATA[628,11] := 19.68756;
   DATA[628,12] := 2.206707;
   DATA[628,13] := 985.4845;
   DATA[628,14] := 1.0;
   DATA[628,15] := 2.0;
   DATA[628,16] := 1.0;
   DATA[628,17] := 1.0;
   DATA[628,18] := 1.0;
   DATA[628,19] := 2.0;
   DATA[628,20] := 148.808;
   DATA[628,21] := 155.7806;
   DATA[628,22] := 1.717105;
   DATA[628,23] := 992.361;
   DATA[628,24] := 2.0;
   DATA[628,25] := 2.0;
   DATA[628,26] := 7.880544;
   DATA[628,27] := 145.1166;
   DATA[628,28] := 263.1377;
   DATA[628,29] := 12.03538;
   DATA[628,30] := 1.726865;
   DATA[628,31] := 1.300756;
   DATA[628,32] := 0.7355248;
   DATA[628,33] := 0.3084265;
   DATA[628,34] := 2.0;
   DATA[628,35] := 250.8972;
   DATA[628,36] := 1.69801;
   DATA[628,37] := 189.5027;
   DATA[628,38] := 0.000128152;
   DATA[628,39] := 1.0;
   DATA[629,0] := 2.451398;
   DATA[629,1] := 536.2319;
   DATA[629,2] := 2.0;
   DATA[629,3] := 2.0;
   DATA[629,4] := 262.1764;
   DATA[629,5] := 8.394514;
   DATA[629,6] := 327.7621;
   DATA[629,7] := 2.439625;
   DATA[629,8] := 2.0;
   DATA[629,9] := 2.0;
   DATA[629,10] := 2.0;
   DATA[629,11] := 19.68756;
   DATA[629,12] := 2.206707;
   DATA[629,13] := 985.4445;
   DATA[629,14] := 1.0;
   DATA[629,15] := 2.0;
   DATA[629,16] := 1.0;
   DATA[629,17] := 1.0;
   DATA[629,18] := 1.0;
   DATA[629,19] := 2.0;
   DATA[629,20] := 148.808;
   DATA[629,21] := 155.7806;
   DATA[629,22] := 1.717105;
   DATA[629,23] := 992.6685;
   DATA[629,24] := 2.0;
   DATA[629,25] := 2.0;
   DATA[629,26] := 7.880544;
   DATA[629,27] := 145.1166;
   DATA[629,28] := 263.1377;
   DATA[629,29] := 12.03538;
   DATA[629,30] := 1.726865;
   DATA[629,31] := 1.302037;
   DATA[629,32] := 0.7355248;
   DATA[629,33] := 0.3084265;
   DATA[629,34] := 2.0;
   DATA[629,35] := 250.8972;
   DATA[629,36] := 1.69801;
   DATA[629,37] := 189.5027;
   DATA[629,38] := 0.000128152;
   DATA[629,39] := 1.0;
   DATA[630,0] := 2.507126;
   DATA[630,1] := 536.0749;
   DATA[630,2] := 2.0;
   DATA[630,3] := 2.0;
   DATA[630,4] := 262.1764;
   DATA[630,5] := 8.396116;
   DATA[630,6] := 327.7621;
   DATA[630,7] := 2.439625;
   DATA[630,8] := 2.0;
   DATA[630,9] := 2.0;
   DATA[630,10] := 2.0;
   DATA[630,11] := 19.65235;
   DATA[630,12] := 2.209653;
   DATA[630,13] := 985.4845;
   DATA[630,14] := 1.0;
   DATA[630,15] := 2.0;
   DATA[630,16] := 1.0;
   DATA[630,17] := 1.0;
   DATA[630,18] := 1.0;
   DATA[630,19] := 2.0;
   DATA[630,20] := 148.808;
   DATA[630,21] := 155.7806;
   DATA[630,22] := 1.717105;
   DATA[630,23] := 992.6685;
   DATA[630,24] := 2.0;
   DATA[630,25] := 2.0;
   DATA[630,26] := 7.878621;
   DATA[630,27] := 145.1166;
   DATA[630,28] := 263.1377;
   DATA[630,29] := 12.03538;
   DATA[630,30] := 1.7293;
   DATA[630,31] := 1.302037;
   DATA[630,32] := 0.7355248;
   DATA[630,33] := 0.3084265;
   DATA[630,34] := 2.0;
   DATA[630,35] := 250.8972;
   DATA[630,36] := 1.69801;
   DATA[630,37] := 189.6148;
   DATA[630,38] := 0.000128152;
   DATA[630,39] := 1.0;
   DATA[631,0] := 2.53467;
   DATA[631,1] := 535.4076;
   DATA[631,2] := 2.0;
   DATA[631,3] := 2.0;
   DATA[631,4] := 262.1764;
   DATA[631,5] := 8.396116;
   DATA[631,6] := 327.7621;
   DATA[631,7] := 2.439625;
   DATA[631,8] := 2.0;
   DATA[631,9] := 2.0;
   DATA[631,10] := 2.0;
   DATA[631,11] := 19.65235;
   DATA[631,12] := 2.209653;
   DATA[631,13] := 985.5646;
   DATA[631,14] := 1.0;
   DATA[631,15] := 2.0;
   DATA[631,16] := 1.0;
   DATA[631,17] := 1.0;
   DATA[631,18] := 1.0;
   DATA[631,19] := 2.0;
   DATA[631,20] := 148.808;
   DATA[631,21] := 155.7806;
   DATA[631,22] := 1.717105;
   DATA[631,23] := 992.7454;
   DATA[631,24] := 2.0;
   DATA[631,25] := 2.0;
   DATA[631,26] := 7.87798;
   DATA[631,27] := 145.1166;
   DATA[631,28] := 263.1377;
   DATA[631,29] := 12.03538;
   DATA[631,30] := 1.7293;
   DATA[631,31] := 1.301012;
   DATA[631,32] := 0.7355248;
   DATA[631,33] := 0.3084265;
   DATA[631,34] := 2.0;
   DATA[631,35] := 250.8972;
   DATA[631,36] := 1.69801;
   DATA[631,37] := 189.6148;
   DATA[631,38] := 0.000128152;
   DATA[631,39] := 1.0;
   DATA[632,0] := 2.578868;
   DATA[632,1] := 535.1329;
   DATA[632,2] := 2.0;
   DATA[632,3] := 2.0;
   DATA[632,4] := 262.1764;
   DATA[632,5] := 8.396116;
   DATA[632,6] := 327.7621;
   DATA[632,7] := 2.441675;
   DATA[632,8] := 2.0;
   DATA[632,9] := 2.0;
   DATA[632,10] := 2.0;
   DATA[632,11] := 19.68756;
   DATA[632,12] := 2.209653;
   DATA[632,13] := 985.6047;
   DATA[632,14] := 1.0;
   DATA[632,15] := 2.0;
   DATA[632,16] := 1.0;
   DATA[632,17] := 1.0;
   DATA[632,18] := 1.0;
   DATA[632,19] := 2.0;
   DATA[632,20] := 148.808;
   DATA[632,21] := 155.7806;
   DATA[632,22] := 1.719156;
   DATA[632,23] := 992.361;
   DATA[632,24] := 2.0;
   DATA[632,25] := 2.0;
   DATA[632,26] := 7.87798;
   DATA[632,27] := 145.1166;
   DATA[632,28] := 263.1377;
   DATA[632,29] := 12.03538;
   DATA[632,30] := 1.731095;
   DATA[632,31] := 1.282439;
   DATA[632,32] := 0.7355248;
   DATA[632,33] := 0.3084265;
   DATA[632,34] := 2.0;
   DATA[632,35] := 250.8972;
   DATA[632,36] := 1.69801;
   DATA[632,37] := 189.6148;
   DATA[632,38] := 0.000128152;
   DATA[632,39] := 1.0;
   DATA[633,0] := 2.608334;
   DATA[633,1] := 534.7403;
   DATA[633,2] := 2.0;
   DATA[633,3] := 2.0;
   DATA[633,4] := 262.1764;
   DATA[633,5] := 8.396116;
   DATA[633,6] := 327.7621;
   DATA[633,7] := 2.441675;
   DATA[633,8] := 2.0;
   DATA[633,9] := 2.0;
   DATA[633,10] := 2.0;
   DATA[633,11] := 19.68756;
   DATA[633,12] := 2.209653;
   DATA[633,13] := 985.4845;
   DATA[633,14] := 1.0;
   DATA[633,15] := 2.0;
   DATA[633,16] := 1.0;
   DATA[633,17] := 1.0;
   DATA[633,18] := 1.0;
   DATA[633,19] := 2.0;
   DATA[633,20] := 148.808;
   DATA[633,21] := 155.7806;
   DATA[633,22] := 1.719156;
   DATA[633,23] := 992.5147;
   DATA[633,24] := 2.0;
   DATA[633,25] := 2.0;
   DATA[633,26] := 7.87798;
   DATA[633,27] := 145.0141;
   DATA[633,28] := 263.1377;
   DATA[633,29] := 12.03538;
   DATA[633,30] := 1.731095;
   DATA[633,31] := 1.281542;
   DATA[633,32] := 0.7355248;
   DATA[633,33] := 0.3084265;
   DATA[633,34] := 2.0;
   DATA[633,35] := 250.8972;
   DATA[633,36] := 1.69801;
   DATA[633,37] := 189.6148;
   DATA[633,38] := 0.000128152;
   DATA[633,39] := 1.0;
   DATA[634,0] := 2.641002;
   DATA[634,1] := 534.6618;
   DATA[634,2] := 2.0;
   DATA[634,3] := 2.0;
   DATA[634,4] := 262.1764;
   DATA[634,5] := 8.396116;
   DATA[634,6] := 327.7621;
   DATA[634,7] := 2.44411;
   DATA[634,8] := 2.0;
   DATA[634,9] := 2.0;
   DATA[634,10] := 2.0;
   DATA[634,11] := 19.68756;
   DATA[634,12] := 2.21324;
   DATA[634,13] := 985.4845;
   DATA[634,14] := 1.0;
   DATA[634,15] := 2.0;
   DATA[634,16] := 1.0;
   DATA[634,17] := 1.0;
   DATA[634,18] := 1.0;
   DATA[634,19] := 2.0;
   DATA[634,20] := 148.808;
   DATA[634,21] := 155.7806;
   DATA[634,22] := 1.719156;
   DATA[634,23] := 992.7454;
   DATA[634,24] := 2.0;
   DATA[634,25] := 2.0;
   DATA[634,26] := 7.87798;
   DATA[634,27] := 144.9628;
   DATA[634,28] := 263.1377;
   DATA[634,29] := 12.03538;
   DATA[634,30] := 1.731095;
   DATA[634,31] := 1.281542;
   DATA[634,32] := 0.7355248;
   DATA[634,33] := 0.3080421;
   DATA[634,34] := 2.0;
   DATA[634,35] := 250.8972;
   DATA[634,36] := 1.69801;
   DATA[634,37] := 189.6148;
   DATA[634,38] := 0.000128152;
   DATA[634,39] := 1.0;
   DATA[635,0] := 2.657656;
   DATA[635,1] := 534.1516;
   DATA[635,2] := 2.0;
   DATA[635,3] := 2.0;
   DATA[635,4] := 262.1764;
   DATA[635,5] := 8.396116;
   DATA[635,6] := 327.7621;
   DATA[635,7] := 2.444366;
   DATA[635,8] := 2.0;
   DATA[635,9] := 2.0;
   DATA[635,10] := 2.0;
   DATA[635,11] := 19.68756;
   DATA[635,12] := 2.21324;
   DATA[635,13] := 985.4845;
   DATA[635,14] := 1.0;
   DATA[635,15] := 2.0;
   DATA[635,16] := 1.0;
   DATA[635,17] := 1.0;
   DATA[635,18] := 1.0;
   DATA[635,19] := 2.0;
   DATA[635,20] := 148.808;
   DATA[635,21] := 155.7806;
   DATA[635,22] := 1.717361;
   DATA[635,23] := 992.707;
   DATA[635,24] := 2.0;
   DATA[635,25] := 2.0;
   DATA[635,26] := 7.87798;
   DATA[635,27] := 144.9628;
   DATA[635,28] := 263.1377;
   DATA[635,29] := 12.03538;
   DATA[635,30] := 1.731095;
   DATA[635,31] := 1.282567;
   DATA[635,32] := 0.7355248;
   DATA[635,33] := 0.3066329;
   DATA[635,34] := 2.0;
   DATA[635,35] := 250.8972;
   DATA[635,36] := 1.69801;
   DATA[635,37] := 189.6148;
   DATA[635,38] := 0.000128152;
   DATA[635,39] := 1.0;
   DATA[636,0] := 2.663741;
   DATA[636,1] := 534.23;
   DATA[636,2] := 2.0;
   DATA[636,3] := 2.0;
   DATA[636,4] := 262.1764;
   DATA[636,5] := 8.396116;
   DATA[636,6] := 327.7621;
   DATA[636,7] := 2.444623;
   DATA[636,8] := 2.0;
   DATA[636,9] := 2.0;
   DATA[636,10] := 2.0;
   DATA[636,11] := 19.68756;
   DATA[636,12] := 2.21324;
   DATA[636,13] := 985.3644;
   DATA[636,14] := 1.0;
   DATA[636,15] := 2.0;
   DATA[636,16] := 1.0;
   DATA[636,17] := 1.0;
   DATA[636,18] := 1.0;
   DATA[636,19] := 2.0;
   DATA[636,20] := 148.808;
   DATA[636,21] := 155.7806;
   DATA[636,22] := 1.717361;
   DATA[636,23] := 992.6685;
   DATA[636,24] := 2.0;
   DATA[636,25] := 2.0;
   DATA[636,26] := 7.87798;
   DATA[636,27] := 144.9628;
   DATA[636,28] := 263.1377;
   DATA[636,29] := 12.03538;
   DATA[636,30] := 1.729172;
   DATA[636,31] := 1.289228;
   DATA[636,32] := 0.7355248;
   DATA[636,33] := 0.3081062;
   DATA[636,34] := 2.0;
   DATA[636,35] := 250.8972;
   DATA[636,36] := 1.69801;
   DATA[636,37] := 189.6148;
   DATA[636,38] := 0.000128152;
   DATA[636,39] := 1.0;
   DATA[637,0] := 2.660539;
   DATA[637,1] := 534.5048;
   DATA[637,2] := 2.0;
   DATA[637,3] := 2.0;
   DATA[637,4] := 262.1764;
   DATA[637,5] := 8.396116;
   DATA[637,6] := 327.7621;
   DATA[637,7] := 2.444623;
   DATA[637,8] := 2.0;
   DATA[637,9] := 2.0;
   DATA[637,10] := 2.0;
   DATA[637,11] := 19.67476;
   DATA[637,12] := 2.21324;
   DATA[637,13] := 985.6047;
   DATA[637,14] := 1.0;
   DATA[637,15] := 2.0;
   DATA[637,16] := 1.0;
   DATA[637,17] := 1.0;
   DATA[637,18] := 1.0;
   DATA[637,19] := 2.0;
   DATA[637,20] := 148.808;
   DATA[637,21] := 155.7806;
   DATA[637,22] := 1.717361;
   DATA[637,23] := 992.5916;
   DATA[637,24] := 2.0;
   DATA[637,25] := 2.0;
   DATA[637,26] := 7.87798;
   DATA[637,27] := 144.9628;
   DATA[637,28] := 263.1377;
   DATA[637,29] := 12.03538;
   DATA[637,30] := 1.729172;
   DATA[637,31] := 1.275266;
   DATA[637,32] := 0.7355248;
   DATA[637,33] := 0.3081062;
   DATA[637,34] := 2.0;
   DATA[637,35] := 250.8972;
   DATA[637,36] := 1.69801;
   DATA[637,37] := 189.6148;
   DATA[637,38] := 0.000128152;
   DATA[637,39] := 1.0;
   DATA[638,0] := 2.628511;
   DATA[638,1] := 534.9366;
   DATA[638,2] := 2.0;
   DATA[638,3] := 2.0;
   DATA[638,4] := 262.1764;
   DATA[638,5] := 8.396116;
   DATA[638,6] := 327.7621;
   DATA[638,7] := 2.443341;
   DATA[638,8] := 2.0;
   DATA[638,9] := 2.0;
   DATA[638,10] := 2.0;
   DATA[638,11] := 19.62354;
   DATA[638,12] := 2.211575;
   DATA[638,13] := 985.6848;
   DATA[638,14] := 1.0;
   DATA[638,15] := 2.0;
   DATA[638,16] := 1.0;
   DATA[638,17] := 1.0;
   DATA[638,18] := 1.0;
   DATA[638,19] := 2.0;
   DATA[638,20] := 148.808;
   DATA[638,21] := 155.7806;
   DATA[638,22] := 1.715567;
   DATA[638,23] := 992.5532;
   DATA[638,24] := 2.0;
   DATA[638,25] := 2.0;
   DATA[638,26] := 7.87798;
   DATA[638,27] := 144.9628;
   DATA[638,28] := 263.1377;
   DATA[638,29] := 12.34299;
   DATA[638,30] := 1.729172;
   DATA[638,31] := 1.261304;
   DATA[638,32] := 0.7355248;
   DATA[638,33] := 0.3081062;
   DATA[638,34] := 2.0;
   DATA[638,35] := 250.8972;
   DATA[638,36] := 1.69801;
   DATA[638,37] := 189.6148;
   DATA[638,38] := 0.000128152;
   DATA[638,39] := 1.0;
   DATA[639,0] := 2.622426;
   DATA[639,1] := 535.2114;
   DATA[639,2] := 2.0;
   DATA[639,3] := 2.0;
   DATA[639,4] := 262.1764;
   DATA[639,5] := 8.396116;
   DATA[639,6] := 327.7621;
   DATA[639,7] := 2.443341;
   DATA[639,8] := 2.0;
   DATA[639,9] := 2.0;
   DATA[639,10] := 2.0;
   DATA[639,11] := 19.60753;
   DATA[639,12] := 2.211447;
   DATA[639,13] := 985.8851;
   DATA[639,14] := 1.0;
   DATA[639,15] := 2.0;
   DATA[639,16] := 1.0;
   DATA[639,17] := 1.0;
   DATA[639,18] := 1.0;
   DATA[639,19] := 2.0;
   DATA[639,20] := 148.808;
   DATA[639,21] := 155.7806;
   DATA[639,22] := 1.715567;
   DATA[639,23] := 992.5532;
   DATA[639,24] := 2.0;
   DATA[639,25] := 2.0;
   DATA[639,26] := 7.87798;
   DATA[639,27] := 144.9628;
   DATA[639,28] := 263.1377;
   DATA[639,29] := 12.34299;
   DATA[639,30] := 1.729172;
   DATA[639,31] := 1.261944;
   DATA[639,32] := 0.7355248;
   DATA[639,33] := 0.3081062;
   DATA[639,34] := 2.0;
   DATA[639,35] := 250.8972;
   DATA[639,36] := 1.617916;
   DATA[639,37] := 189.6148;
   DATA[639,38] := 0.000128152;
   DATA[639,39] := 1.0;
   DATA[640,0] := 2.616981;
   DATA[640,1] := 535.2114;
   DATA[640,2] := 2.0;
   DATA[640,3] := 2.0;
   DATA[640,4] := 262.1764;
   DATA[640,5] := 8.395155;
   DATA[640,6] := 327.7621;
   DATA[640,7] := 2.443341;
   DATA[640,8] := 2.0;
   DATA[640,9] := 2.0;
   DATA[640,10] := 2.0;
   DATA[640,11] := 19.57872;
   DATA[640,12] := 2.211447;
   DATA[640,13] := 985.7649;
   DATA[640,14] := 1.0;
   DATA[640,15] := 2.0;
   DATA[640,16] := 1.0;
   DATA[640,17] := 1.0;
   DATA[640,18] := 1.0;
   DATA[640,19] := 2.0;
   DATA[640,20] := 148.808;
   DATA[640,21] := 155.7806;
   DATA[640,22] := 1.715567;
   DATA[640,23] := 992.7839;
   DATA[640,24] := 2.0;
   DATA[640,25] := 2.0;
   DATA[640,26] := 7.87798;
   DATA[640,27] := 144.9628;
   DATA[640,28] := 263.1377;
   DATA[640,29] := 12.34299;
   DATA[640,30] := 1.729172;
   DATA[640,31] := 1.280902;
   DATA[640,32] := 0.7355248;
   DATA[640,33] := 0.3081062;
   DATA[640,34] := 2.0;
   DATA[640,35] := 250.8972;
   DATA[640,36] := 1.617916;
   DATA[640,37] := 189.6148;
   DATA[640,38] := 0.000128152;
   DATA[640,39] := 1.0;
   DATA[641,0] := 2.601287;
   DATA[641,1] := 535.3291;
   DATA[641,2] := 2.0;
   DATA[641,3] := 2.0;
   DATA[641,4] := 262.1764;
   DATA[641,5] := 8.395155;
   DATA[641,6] := 327.7621;
   DATA[641,7] := 2.443341;
   DATA[641,8] := 2.0;
   DATA[641,9] := 2.0;
   DATA[641,10] := 2.0;
   DATA[641,11] := 19.5275;
   DATA[641,12] := 2.211447;
   DATA[641,13] := 986.0052;
   DATA[641,14] := 1.0;
   DATA[641,15] := 2.0;
   DATA[641,16] := 1.0;
   DATA[641,17] := 1.0;
   DATA[641,18] := 1.0;
   DATA[641,19] := 2.0;
   DATA[641,20] := 148.808;
   DATA[641,21] := 155.7806;
   DATA[641,22] := 1.715567;
   DATA[641,23] := 992.8608;
   DATA[641,24] := 2.0;
   DATA[641,25] := 2.0;
   DATA[641,26] := 7.87798;
   DATA[641,27] := 144.9628;
   DATA[641,28] := 263.1377;
   DATA[641,29] := 12.15073;
   DATA[641,30] := 1.729172;
   DATA[641,31] := 1.28167;
   DATA[641,32] := 0.7355248;
   DATA[641,33] := 0.3081062;
   DATA[641,34] := 2.0;
   DATA[641,35] := 250.8972;
   DATA[641,36] := 1.617916;
   DATA[641,37] := 189.6148;
   DATA[641,38] := 0.000128152;
   DATA[641,39] := 1.0;
   DATA[642,0] := 2.585914;
   DATA[642,1] := 535.4469;
   DATA[642,2] := 2.0;
   DATA[642,3] := 2.0;
   DATA[642,4] := 262.1764;
   DATA[642,5] := 8.395155;
   DATA[642,6] := 327.7621;
   DATA[642,7] := 2.440393;
   DATA[642,8] := 2.0;
   DATA[642,9] := 2.0;
   DATA[642,10] := 2.0;
   DATA[642,11] := 19.5275;
   DATA[642,12] := 2.211447;
   DATA[642,13] := 986.0853;
   DATA[642,14] := 1.0;
   DATA[642,15] := 2.0;
   DATA[642,16] := 1.0;
   DATA[642,17] := 1.0;
   DATA[642,18] := 1.0;
   DATA[642,19] := 2.0;
   DATA[642,20] := 148.808;
   DATA[642,21] := 155.7806;
   DATA[642,22] := 1.715567;
   DATA[642,23] := 992.9761;
   DATA[642,24] := 2.0;
   DATA[642,25] := 2.0;
   DATA[642,26] := 7.878942;
   DATA[642,27] := 144.9628;
   DATA[642,28] := 263.1377;
   DATA[642,29] := 12.03538;
   DATA[642,30] := 1.729172;
   DATA[642,31] := 1.28167;
   DATA[642,32] := 0.7339884;
   DATA[642,33] := 0.3084905;
   DATA[642,34] := 2.0;
   DATA[642,35] := 250.8972;
   DATA[642,36] := 1.617916;
   DATA[642,37] := 189.6148;
   DATA[642,38] := 0.000128152;
   DATA[642,39] := 1.0;
   DATA[643,0] := 2.564456;
   DATA[643,1] := 535.8394;
   DATA[643,2] := 2.0;
   DATA[643,3] := 2.0;
   DATA[643,4] := 262.1764;
   DATA[643,5] := 8.395155;
   DATA[643,6] := 327.7621;
   DATA[643,7] := 2.439753;
   DATA[643,8] := 2.0;
   DATA[643,9] := 2.0;
   DATA[643,10] := 2.0;
   DATA[643,11] := 19.5275;
   DATA[643,12] := 2.211447;
   DATA[643,13] := 986.0853;
   DATA[643,14] := 1.0;
   DATA[643,15] := 2.0;
   DATA[643,16] := 1.0;
   DATA[643,17] := 1.0;
   DATA[643,18] := 1.0;
   DATA[643,19] := 2.0;
   DATA[643,20] := 148.808;
   DATA[643,21] := 155.7806;
   DATA[643,22] := 1.715567;
   DATA[643,23] := 993.053;
   DATA[643,24] := 2.0;
   DATA[643,25] := 2.0;
   DATA[643,26] := 7.878942;
   DATA[643,27] := 144.9628;
   DATA[643,28] := 263.1377;
   DATA[643,29] := 12.03538;
   DATA[643,30] := 1.730838;
   DATA[643,31] := 1.277956;
   DATA[643,32] := 0.7339884;
   DATA[643,33] := 0.3084905;
   DATA[643,34] := 2.0;
   DATA[643,35] := 250.8972;
   DATA[643,36] := 1.617916;
   DATA[643,37] := 189.6148;
   DATA[643,38] := 0.000128152;
   DATA[643,39] := 1.0;
   DATA[644,0] := 2.548762;
   DATA[644,1] := 535.6431;
   DATA[644,2] := 2.0;
   DATA[644,3] := 2.0;
   DATA[644,4] := 262.1764;
   DATA[644,5] := 8.395155;
   DATA[644,6] := 327.7621;
   DATA[644,7] := 2.439753;
   DATA[644,8] := 2.0;
   DATA[644,9] := 2.0;
   DATA[644,10] := 2.0;
   DATA[644,11] := 19.59793;
   DATA[644,12] := 2.210166;
   DATA[644,13] := 986.2856;
   DATA[644,14] := 1.0;
   DATA[644,15] := 2.0;
   DATA[644,16] := 1.0;
   DATA[644,17] := 1.0;
   DATA[644,18] := 1.0;
   DATA[644,19] := 2.0;
   DATA[644,20] := 148.808;
   DATA[644,21] := 155.7806;
   DATA[644,22] := 1.715567;
   DATA[644,23] := 993.0915;
   DATA[644,24] := 2.0;
   DATA[644,25] := 2.0;
   DATA[644,26] := 7.878942;
   DATA[644,27] := 144.9628;
   DATA[644,28] := 263.1697;
   DATA[644,29] := 12.03538;
   DATA[644,30] := 1.730838;
   DATA[644,31] := 1.275266;
   DATA[644,32] := 0.7360369;
   DATA[644,33] := 0.3084905;
   DATA[644,34] := 2.0;
   DATA[644,35] := 250.8011;
   DATA[644,36] := 1.762086;
   DATA[644,37] := 189.5668;
   DATA[644,38] := 0.000128152;
   DATA[644,39] := 1.0;
   DATA[645,0] := 2.533068;
   DATA[645,1] := 535.2506;
   DATA[645,2] := 2.0;
   DATA[645,3] := 2.0;
   DATA[645,4] := 262.1764;
   DATA[645,5] := 8.395155;
   DATA[645,6] := 327.7621;
   DATA[645,7] := 2.439753;
   DATA[645,8] := 2.0;
   DATA[645,9] := 2.0;
   DATA[645,10] := 2.0;
   DATA[645,11] := 19.62674;
   DATA[645,12] := 2.210166;
   DATA[645,13] := 986.6461;
   DATA[645,14] := 1.0;
   DATA[645,15] := 2.0;
   DATA[645,16] := 1.0;
   DATA[645,17] := 1.0;
   DATA[645,18] := 1.0;
   DATA[645,19] := 2.0;
   DATA[645,20] := 148.808;
   DATA[645,21] := 155.7806;
   DATA[645,22] := 1.714798;
   DATA[645,23] := 992.9761;
   DATA[645,24] := 2.0;
   DATA[645,25] := 2.0;
   DATA[645,26] := 7.878942;
   DATA[645,27] := 144.9628;
   DATA[645,28] := 263.4261;
   DATA[645,29] := 12.03538;
   DATA[645,30] := 1.730838;
   DATA[645,31] := 1.289484;
   DATA[645,32] := 0.7360369;
   DATA[645,33] := 0.3074016;
   DATA[645,34] := 2.0;
   DATA[645,35] := 250.6569;
   DATA[645,36] := 1.762086;
   DATA[645,37] := 189.5347;
   DATA[645,38] := 0.000128152;
   DATA[645,39] := 1.0;
   DATA[646,0] := 2.517695;
   DATA[646,1] := 534.8973;
   DATA[646,2] := 2.0;
   DATA[646,3] := 2.0;
   DATA[646,4] := 262.1764;
   DATA[646,5] := 8.395155;
   DATA[646,6] := 327.7621;
   DATA[646,7] := 2.439753;
   DATA[646,8] := 2.0;
   DATA[646,9] := 2.0;
   DATA[646,10] := 2.0;
   DATA[646,11] := 19.62674;
   DATA[646,12] := 2.210166;
   DATA[646,13] := 987.0466;
   DATA[646,14] := 1.0;
   DATA[646,15] := 2.0;
   DATA[646,16] := 1.0;
   DATA[646,17] := 1.0;
   DATA[646,18] := 1.0;
   DATA[646,19] := 2.0;
   DATA[646,20] := 148.808;
   DATA[646,21] := 155.7806;
   DATA[646,22] := 1.714542;
   DATA[646,23] := 993.053;
   DATA[646,24] := 2.0;
   DATA[646,25] := 2.0;
   DATA[646,26] := 7.878942;
   DATA[646,27] := 145.1166;
   DATA[646,28] := 263.4261;
   DATA[646,29] := 12.03538;
   DATA[646,30] := 1.727634;
   DATA[646,31] := 1.300756;
   DATA[646,32] := 0.7360369;
   DATA[646,33] := 0.3068251;
   DATA[646,34] := 2.0;
   DATA[646,35] := 250.6569;
   DATA[646,36] := 1.762086;
   DATA[646,37] := 189.5027;
   DATA[646,38] := 0.000128152;
   DATA[646,39] := 1.0;
   DATA[647,0] := 2.498799;
   DATA[647,1] := 534.6226;
   DATA[647,2] := 2.0;
   DATA[647,3] := 2.0;
   DATA[647,4] := 262.1764;
   DATA[647,5] := 8.395155;
   DATA[647,6] := 327.7621;
   DATA[647,7] := 2.439753;
   DATA[647,8] := 2.0;
   DATA[647,9] := 2.0;
   DATA[647,10] := 2.0;
   DATA[647,11] := 19.62674;
   DATA[647,12] := 2.211447;
   DATA[647,13] := 987.4471;
   DATA[647,14] := 1.0;
   DATA[647,15] := 2.0;
   DATA[647,16] := 1.0;
   DATA[647,17] := 1.0;
   DATA[647,18] := 1.0;
   DATA[647,19] := 2.0;
   DATA[647,20] := 148.808;
   DATA[647,21] := 155.7806;
   DATA[647,22] := 1.714542;
   DATA[647,23] := 992.8992;
   DATA[647,24] := 2.0;
   DATA[647,25] := 2.0;
   DATA[647,26] := 7.878942;
   DATA[647,27] := 145.1166;
   DATA[647,28] := 263.4261;
   DATA[647,29] := 12.03538;
   DATA[647,30] := 1.727634;
   DATA[647,31] := 1.297554;
   DATA[647,32] := 0.7360369;
   DATA[647,33] := 0.3068251;
   DATA[647,34] := 2.0;
   DATA[647,35] := 250.6569;
   DATA[647,36] := 1.601897;
   DATA[647,37] := 189.3745;
   DATA[647,38] := 0.000128152;
   DATA[647,39] := 1.0;
   DATA[648,0] := 2.483426;
   DATA[648,1] := 534.3085;
   DATA[648,2] := 2.0;
   DATA[648,3] := 2.0;
   DATA[648,4] := 262.1764;
   DATA[648,5] := 8.395155;
   DATA[648,6] := 327.7621;
   DATA[648,7] := 2.439753;
   DATA[648,8] := 2.0;
   DATA[648,9] := 2.0;
   DATA[648,10] := 2.0;
   DATA[648,11] := 19.66835;
   DATA[648,12] := 2.211447;
   DATA[648,13] := 987.0867;
   DATA[648,14] := 1.0;
   DATA[648,15] := 2.0;
   DATA[648,16] := 1.0;
   DATA[648,17] := 1.0;
   DATA[648,18] := 1.0;
   DATA[648,19] := 2.0;
   DATA[648,20] := 148.808;
   DATA[648,21] := 155.7806;
   DATA[648,22] := 1.715824;
   DATA[648,23] := 993.2453;
   DATA[648,24] := 2.0;
   DATA[648,25] := 2.0;
   DATA[648,26] := 7.878942;
   DATA[648,27] := 145.1166;
   DATA[648,28] := 263.4261;
   DATA[648,29] := 12.03538;
   DATA[648,30] := 1.727634;
   DATA[648,31] := 1.291918;
   DATA[648,32] := 0.7346286;
   DATA[648,33] := 0.3068251;
   DATA[648,34] := 2.0;
   DATA[648,35] := 250.6569;
   DATA[648,36] := 1.601897;
   DATA[648,37] := 189.3745;
   DATA[648,38] := 0.000128152;
   DATA[648,39] := 1.0;
   DATA[649,0] := 2.463248;
   DATA[649,1] := 534.6226;
   DATA[649,2] := 2.0;
   DATA[649,3] := 2.0;
   DATA[649,4] := 262.1764;
   DATA[649,5] := 8.395155;
   DATA[649,6] := 327.7621;
   DATA[649,7] := 2.439753;
   DATA[649,8] := 2.0;
   DATA[649,9] := 2.0;
   DATA[649,10] := 2.0;
   DATA[649,11] := 19.57552;
   DATA[649,12] := 2.211447;
   DATA[649,13] := 987.2068;
   DATA[649,14] := 1.0;
   DATA[649,15] := 2.0;
   DATA[649,16] := 1.0;
   DATA[649,17] := 1.0;
   DATA[649,18] := 1.0;
   DATA[649,19] := 2.0;
   DATA[649,20] := 148.808;
   DATA[649,21] := 155.7806;
   DATA[649,22] := 1.716849;
   DATA[649,23] := 993.2453;
   DATA[649,24] := 2.0;
   DATA[649,25] := 2.0;
   DATA[649,26] := 7.878942;
   DATA[649,27] := 145.1166;
   DATA[649,28] := 263.1697;
   DATA[649,29] := 12.03538;
   DATA[649,30] := 1.727634;
   DATA[649,31] := 1.281927;
   DATA[649,32] := 0.7346286;
   DATA[649,33] := 0.3066329;
   DATA[649,34] := 2.0;
   DATA[649,35] := 250.6569;
   DATA[649,36] := 1.601897;
   DATA[649,37] := 189.3745;
   DATA[649,38] := 0.000128152;
   DATA[649,39] := 1.0;
   DATA[650,0] := 2.463248;
   DATA[650,1] := 534.6226;
   DATA[650,2] := 2.0;
   DATA[650,3] := 2.0;
   DATA[650,4] := 262.1764;
   DATA[650,5] := 8.395155;
   DATA[650,6] := 327.7621;
   DATA[650,7] := 2.439753;
   DATA[650,8] := 2.0;
   DATA[650,9] := 2.0;
   DATA[650,10] := 2.0;
   DATA[650,11] := 19.57552;
   DATA[650,12] := 2.211447;
   DATA[650,13] := 987.2068;
   DATA[650,14] := 1.0;
   DATA[650,15] := 2.0;
   DATA[650,16] := 1.0;
   DATA[650,17] := 1.0;
   DATA[650,18] := 1.0;
   DATA[650,19] := 2.0;
   DATA[650,20] := 148.808;
   DATA[650,21] := 155.7806;
   DATA[650,22] := 1.716849;
   DATA[650,23] := 993.2453;
   DATA[650,24] := 2.0;
   DATA[650,25] := 2.0;
   DATA[650,26] := 7.878942;
   DATA[650,27] := 145.1166;
   DATA[650,28] := 263.1697;
   DATA[650,29] := 12.03538;
   DATA[650,30] := 1.727634;
   DATA[650,31] := 1.281927;
   DATA[650,32] := 0.7346286;
   DATA[650,33] := 0.3066329;
   DATA[650,34] := 2.0;
   DATA[650,35] := 250.6569;
   DATA[650,36] := 1.601897;
   DATA[650,37] := 189.3745;
   DATA[650,38] := 0.000128152;
   DATA[650,39] := 1.0;
   DATA[651,0] := 2.447234;
   DATA[651,1] := 534.701;
   DATA[651,2] := 2.0;
   DATA[651,3] := 2.0;
   DATA[651,4] := 262.1764;
   DATA[651,5] := 8.395155;
   DATA[651,6] := 327.7621;
   DATA[651,7] := 2.439753;
   DATA[651,8] := 2.0;
   DATA[651,9] := 2.0;
   DATA[651,10] := 2.0;
   DATA[651,11] := 19.57552;
   DATA[651,12] := 2.212856;
   DATA[651,13] := 987.0065;
   DATA[651,14] := 1.0;
   DATA[651,15] := 2.0;
   DATA[651,16] := 1.0;
   DATA[651,17] := 1.0;
   DATA[651,18] := 1.0;
   DATA[651,19] := 2.0;
   DATA[651,20] := 148.808;
   DATA[651,21] := 155.7806;
   DATA[651,22] := 1.717361;
   DATA[651,23] := 993.1684;
   DATA[651,24] := 2.0;
   DATA[651,25] := 2.0;
   DATA[651,26] := 7.878942;
   DATA[651,27] := 145.1166;
   DATA[651,28] := 263.1697;
   DATA[651,29] := 12.03538;
   DATA[651,30] := 1.727634;
   DATA[651,31] := 1.281158;
   DATA[651,32] := 0.7346286;
   DATA[651,33] := 0.3066329;
   DATA[651,34] := 2.0;
   DATA[651,35] := 250.8331;
   DATA[651,36] := 1.601897;
   DATA[651,37] := 189.6629;
   DATA[651,38] := 0.000128152;
   DATA[651,39] := 1.0;
   DATA[652,0] := 2.431861;
   DATA[652,1] := 535.9179;
   DATA[652,2] := 2.0;
   DATA[652,3] := 2.0;
   DATA[652,4] := 262.1764;
   DATA[652,5] := 8.395155;
   DATA[652,6] := 327.7621;
   DATA[652,7] := 2.44206;
   DATA[652,8] := 2.0;
   DATA[652,9] := 2.0;
   DATA[652,10] := 2.0;
   DATA[652,11] := 19.57552;
   DATA[652,12] := 2.212856;
   DATA[652,13] := 987.0466;
   DATA[652,14] := 1.0;
   DATA[652,15] := 2.0;
   DATA[652,16] := 1.0;
   DATA[652,17] := 1.0;
   DATA[652,18] := 1.0;
   DATA[652,19] := 2.0;
   DATA[652,20] := 148.808;
   DATA[652,21] := 155.7806;
   DATA[652,22] := 1.719284;
   DATA[652,23] := 993.3607;
   DATA[652,24] := 2.0;
   DATA[652,25] := 2.0;
   DATA[652,26] := 7.878942;
   DATA[652,27] := 145.1166;
   DATA[652,28] := 263.1697;
   DATA[652,29] := 12.03538;
   DATA[652,30] := 1.725968;
   DATA[652,31] := 1.289356;
   DATA[652,32] := 0.7361649;
   DATA[652,33] := 0.3066329;
   DATA[652,34] := 2.0;
   DATA[652,35] := 250.8331;
   DATA[652,36] := 1.601897;
   DATA[652,37] := 189.6629;
   DATA[652,38] := 0.000128152;
   DATA[652,39] := 1.0;
   DATA[653,0] := 2.428979;
   DATA[653,1] := 537.017;
   DATA[653,2] := 2.0;
   DATA[653,3] := 2.0;
   DATA[653,4] := 262.1764;
   DATA[653,5] := 8.395155;
   DATA[653,6] := 327.7621;
   DATA[653,7] := 2.44206;
   DATA[653,8] := 2.0;
   DATA[653,9] := 2.0;
   DATA[653,10] := 2.0;
